//     Term 23 (AT2000-0250)/CC Outputs/Current setpoint value Ch.15 <-> Data Pointer/CurrentSetpointValues[14]
//     Term 23 (AT2000-0250)/CC Outputs/Current setpoint value Ch.2 <-> Data Pointer/CurrentSetpointValues[1]
//     Term 23 (AT2000-0250)/CC Outputs/Current setpoint value Ch.3 <-> Data Pointer/CurrentSetpointValues[2]
//     Term 23 (AT2000-0250)/CC Outputs/Current setpoint value Ch.4 <-> Data Pointer/CurrentSetpointValues[3]
//     Term 23 (AT2000-0250)/CC Outputs/Current setpoint value Ch.5 <-> Data Pointer/CurrentSetpointValues[4]
//     Term 23 (AT2000-0250)/CC Outputs/Current setpoint value Ch.6 <-> Data Pointer/CurrentSetpointValues[5]
//     Term 23 (AT2000-0250)/CC Outputs/Current setpoint value Ch.7 <-> Data Pointer/CurrentSetpointValues[6]
//     Term 23 (AT2000-0250)/CC Outputs/Current setpoint value Ch.8 <-> Data Pointer/CurrentSetpointValues[7]
//     Term 23 (AT2000-0250)/CC Outputs/Current setpoint value Ch.9 <-> Data Pointer/CurrentSetpointValues[8]
//     Term 23 (AT2000-0250)/Term 24 (AT2000-5250)/FB Inputs/Value Channel 01 <-> Data Pointer/RawPositionValues[0]
//     Term 23 (AT2000-0250)/Term 24 (AT2000-5250)/FB Inputs/Value Channel 02 <-> Data Pointer/RawPositionValues[1]
//     Term 23 (AT2000-0250)/Term 24 (AT2000-5250)/FB Inputs/Value Channel 03 <-> Data Pointer/RawPositionValues[2]
//     Term 23 (AT2000-0250)/Term 24 (AT2000-5250)/FB Inputs/Value Channel 04 <-> Data Pointer/RawPositionValues[3]
//     Term 23 (AT2000-0250)/Term 24 (AT2000-5250)/FB Inputs/Value Channel 05 <-> Data Pointer/RawPositionValues[4]
//     Term 23 (AT2000-0250)/Term 24 (AT2000-5250)/FB Inputs/Value Channel 06 <-> Data Pointer/RawPositionValues[5]
//     Term 23 (AT2000-0250)/Term 24 (AT2000-5250)/FB Inputs/Value Channel 07 <-> Data Pointer/RawPositionValues[6]
//     Term 23 (AT2000-0250)/Term 24 (AT2000-5250)/FB Inputs/Value Channel 08 <-> Data Pointer/RawPositionValues[7]
//     Term 23 (AT2000-0250)/Term 24 (AT2000-5250)/FB Inputs/Value Channel 09 <-> Data Pointer/RawPositionValues[8]
//     Term 23 (AT2000-0250)/Term 24 (AT2000-5250)/FB Inputs/Value Channel 10 <-> Data Pointer/RawPositionValues[9]
//     Term 23 (AT2000-0250)/Term 24 (AT2000-5250)/FB Inputs/Value Channel 11 <-> Data Pointer/RawPositionValues[10]
//     Term 23 (AT2000-0250)/Term 24 (AT2000-5250)/FB Inputs/Value Channel 12 <-> Data Pointer/RawPositionValues[11]
//     Term 23 (AT2000-0250)/Term 24 (AT2000-5250)/FB Inputs/Value Channel 13 <-> Data Pointer/RawPositionValues[12]
//     Term 23 (AT2000-0250)/Term 24 (AT2000-5250)/FB Inputs/Value Channel 14 <-> Data Pointer/RawPositionValues[13]
//     Term 23 (AT2000-0250)/Term 24 (AT2000-5250)/FB Inputs/Value Channel 15 <-> Data Pointer/RawPositionValues[14]
//     Term 23 (AT2000-0250)/Term 24 (AT2000-5250)/FB Inputs/Value Channel 16 <-> Data Pointer/RawPositionValues[15]
//     Term 23 (AT2000-0250)/Term 24 (AT2000-5250)/FB Inputs/Value Channel 17 <-> Data Pointer/RawPositionValues[16]
//     Term 23 (AT2000-0250)/Term 24 (AT2000-5250)/FB Inputs/Value Channel 18 <-> Data Pointer/RawPositionValues[17]
//     Term 23 (AT2000-0250)/Term 24 (AT2000-5250)/FB Inputs/Value Channel 19 <-> Data Pointer/RawPositionValues[18]
//     Term 23 (AT2000-0250)/Term 24 (AT2000-5250)/FB Inputs/Value Channel 20 <-> Data Pointer/RawPositionValues[19]
//     Term 23 (AT2000-0250)/Term 24 (AT2000-5250)/FB Inputs/Value Channel 21 <-> Data Pointer/RawPositionValues[20]
//     Term 23 (AT2000-0250)/Term 24 (AT2000-5250)/FB Inputs/Value Channel 22 <-> Data Pointer/RawPositionValues[21]
//     Term 23 (AT2000-0250)/Term 24 (AT2000-5250)/FB Inputs/Value Channel 23 <-> Data Pointer/RawPositionValues[22]
//     Term 23 (AT2000-0250)/Term 24 (AT2000-5250)/FB Inputs/Value Channel 24 <-> Data Pointer/RawPositionValues[23]
//     Term 23 (AT2000-0250)/Term 24 (AT2000-5250)/FB Inputs/Value Channel 25 <-> Data Pointer/RawPositionValues[24]
//     Term 23 (AT2000-0250)/Term 24 (AT2000-5250)/FB Inputs/Value Channel 26 <-> Data Pointer/RawPositionValues[25]
//     Term 23 (AT2000-0250)/Term 24 (AT2000-5250)/FB Inputs/Value Channel 27 <-> Data Pointer/RawPositionValues[26]
//     Term 23 (AT2000-0250)/Term 24 (AT2000-5250)/FB Inputs/Value Channel 28 <-> Data Pointer/RawPositionValues[27]
//     Term 23 (AT2000-0250)/Term 24 (AT2000-5250)/FB Inputs/Value Channel 29 <-> Data Pointer/RawPositionValues[28]
//     Term 23 (AT2000-0250)/Term 24 (AT2000-5250)/FB Inputs/Value Channel 30 <-> Data Pointer/RawPositionValues[29]
//     Term 23 (AT2000-0250)/Term 24 (AT2000-5250)/FB Inputs/Value Channel 31 <-> Data Pointer/RawPositionValues[30]
//     Term 23 (AT2000-0250)/Term 24 (AT2000-5250)/FB Inputs/Value Channel 32 <-> Data Pointer/RawPositionValues[31]
//   Device 16 <-> TcCOM Objects/XTS ProcessingUnit 1/Part 1/Module 7
//     Term 13 (AT2002-0250)/CC Inputs/Current actual value Ch.1 <-> Data Pointer/CurrentActualValues[0]
//     Term 13 (AT2002-0250)/CC Inputs/Current actual value Ch.10 <-> Data Pointer/CurrentActualValues[9]
//     Term 13 (AT2002-0250)/CC Inputs/Current actual value Ch.11 <-> Data Pointer/CurrentActualValues[10]
//     Term 13 (AT2002-0250)/CC Inputs/Current actual value Ch.12 <-> Data Pointer/CurrentActualValues[11]
//     Term 13 (AT2002-0250)/CC Inputs/Current actual value Ch.13 <-> Data Pointer/CurrentActualValues[12]
//     Term 13 (AT2002-0250)/CC Inputs/Current actual value Ch.14 <-> Data Pointer/CurrentActualValues[13]
//     Term 13 (AT2002-0250)/CC Inputs/Current actual value Ch.15 <-> Data Pointer/CurrentActualValues[14]
//     Term 13 (AT2002-0250)/CC Inputs/Current actual value Ch.2 <-> Data Pointer/CurrentActualValues[1]
//     Term 13 (AT2002-0250)/CC Inputs/Current actual value Ch.3 <-> Data Pointer/CurrentActualValues[2]
//     Term 13 (AT2002-0250)/CC Inputs/Current actual value Ch.4 <-> Data Pointer/CurrentActualValues[3]
//     Term 13 (AT2002-0250)/CC Inputs/Current actual value Ch.5 <-> Data Pointer/CurrentActualValues[4]
//     Term 13 (AT2002-0250)/CC Inputs/Current actual value Ch.6 <-> Data Pointer/CurrentActualValues[5]
//     Term 13 (AT2002-0250)/CC Inputs/Current actual value Ch.7 <-> Data Pointer/CurrentActualValues[6]
//     Term 13 (AT2002-0250)/CC Inputs/Current actual value Ch.8 <-> Data Pointer/CurrentActualValues[7]
//     Term 13 (AT2002-0250)/CC Inputs/Current actual value Ch.9 <-> Data Pointer/CurrentActualValues[8]
//     Term 13 (AT2002-0250)/CC Inputs/Status <-> Data Pointer/Status
//     Term 13 (AT2002-0250)/CC Outputs/Control <-> Data Pointer/Control
//     Term 13 (AT2002-0250)/CC Outputs/Current setpoint value Ch.1 <-> Data Pointer/CurrentSetpointValues[0]
//     Term 13 (AT2002-0250)/CC Outputs/Current setpoint value Ch.10 <-> Data Pointer/CurrentSetpointValues[9]
//     Term 13 (AT2002-0250)/CC Outputs/Current setpoint value Ch.11 <-> Data Pointer/CurrentSetpointValues[10]
//     Term 13 (AT2002-0250)/CC Outputs/Current setpoint value Ch.12 <-> Data Pointer/CurrentSetpointValues[11]
//     Term 13 (AT2002-0250)/CC Outputs/Current setpoint value Ch.13 <-> Data Pointer/CurrentSetpointValues[12]
//     Term 13 (AT2002-0250)/CC Outputs/Current setpoint value Ch.14 <-> Data Pointer/CurrentSetpointValues[13]
//     Term 13 (AT2002-0250)/CC Outputs/Current setpoint value Ch.15 <-> Data Pointer/CurrentSetpointValues[14]
//     Term 13 (AT2002-0250)/CC Outputs/Current setpoint value Ch.2 <-> Data Pointer/CurrentSetpointValues[1]
//     Term 13 (AT2002-0250)/CC Outputs/Current setpoint value Ch.3 <-> Data Pointer/CurrentSetpointValues[2]
//     Term 13 (AT2002-0250)/CC Outputs/Current setpoint value Ch.4 <-> Data Pointer/CurrentSetpointValues[3]
//     Term 13 (AT2002-0250)/CC Outputs/Current setpoint value Ch.5 <-> Data Pointer/CurrentSetpointValues[4]
//     Term 13 (AT2002-0250)/CC Outputs/Current setpoint value Ch.6 <-> Data Pointer/CurrentSetpointValues[5]
//     Term 13 (AT2002-0250)/CC Outputs/Current setpoint value Ch.7 <-> Data Pointer/CurrentSetpointValues[6]
//     Term 13 (AT2002-0250)/CC Outputs/Current setpoint value Ch.8 <-> Data Pointer/CurrentSetpointValues[7]
//     Term 13 (AT2002-0250)/CC Outputs/Current setpoint value Ch.9 <-> Data Pointer/CurrentSetpointValues[8]
//     Term 13 (AT2002-0250)/Term 14 (AT2002-5250)/FB Inputs/Value Channel 01 <-> Data Pointer/RawPositionValues[0]
//     Term 13 (AT2002-0250)/Term 14 (AT2002-5250)/FB Inputs/Value Channel 02 <-> Data Pointer/RawPositionValues[1]
//     Term 13 (AT2002-0250)/Term 14 (AT2002-5250)/FB Inputs/Value Channel 03 <-> Data Pointer/RawPositionValues[2]
//     Term 13 (AT2002-0250)/Term 14 (AT2002-5250)/FB Inputs/Value Channel 04 <-> Data Pointer/RawPositionValues[3]
//     Term 13 (AT2002-0250)/Term 14 (AT2002-5250)/FB Inputs/Value Channel 05 <-> Data Pointer/RawPositionValues[4]
//     Term 13 (AT2002-0250)/Term 14 (AT2002-5250)/FB Inputs/Value Channel 06 <-> Data Pointer/RawPositionValues[5]
//     Term 13 (AT2002-0250)/Term 14 (AT2002-5250)/FB Inputs/Value Channel 07 <-> Data Pointer/RawPositionValues[6]
//     Term 13 (AT2002-0250)/Term 14 (AT2002-5250)/FB Inputs/Value Channel 08 <-> Data Pointer/RawPositionValues[7]
//     Term 13 (AT2002-0250)/Term 14 (AT2002-5250)/FB Inputs/Value Channel 09 <-> Data Pointer/RawPositionValues[8]
//     Term 13 (AT2002-0250)/Term 14 (AT2002-5250)/FB Inputs/Value Channel 10 <-> Data Pointer/RawPositionValues[9]
//     Term 13 (AT2002-0250)/Term 14 (AT2002-5250)/FB Inputs/Value Channel 11 <-> Data Pointer/RawPositionValues[10]
//     Term 13 (AT2002-0250)/Term 14 (AT2002-5250)/FB Inputs/Value Channel 12 <-> Data Pointer/RawPositionValues[11]
//     Term 13 (AT2002-0250)/Term 14 (AT2002-5250)/FB Inputs/Value Channel 13 <-> Data Pointer/RawPositionValues[12]
//     Term 13 (AT2002-0250)/Term 14 (AT2002-5250)/FB Inputs/Value Channel 14 <-> Data Pointer/RawPositionValues[13]
//     Term 13 (AT2002-0250)/Term 14 (AT2002-5250)/FB Inputs/Value Channel 15 <-> Data Pointer/RawPositionValues[14]
//     Term 13 (AT2002-0250)/Term 14 (AT2002-5250)/FB Inputs/Value Channel 16 <-> Data Pointer/RawPositionValues[15]
//     Term 13 (AT2002-0250)/Term 14 (AT2002-5250)/FB Inputs/Value Channel 17 <-> Data Pointer/RawPositionValues[16]
//     Term 13 (AT2002-0250)/Term 14 (AT2002-5250)/FB Inputs/Value Channel 18 <-> Data Pointer/RawPositionValues[17]
//     Term 13 (AT2002-0250)/Term 14 (AT2002-5250)/FB Inputs/Value Channel 19 <-> Data Pointer/RawPositionValues[18]
//     Term 13 (AT2002-0250)/Term 14 (AT2002-5250)/FB Inputs/Value Channel 20 <-> Data Pointer/RawPositionValues[19]
//     Term 13 (AT2002-0250)/Term 14 (AT2002-5250)/FB Inputs/Value Channel 21 <-> Data Pointer/RawPositionValues[20]
//     Term 13 (AT2002-0250)/Term 14 (AT2002-5250)/FB Inputs/Value Channel 22 <-> Data Pointer/RawPositionValues[21]
//     Term 13 (AT2002-0250)/Term 14 (AT2002-5250)/FB Inputs/Value Channel 23 <-> Data Pointer/RawPositionValues[22]
//     Term 13 (AT2002-0250)/Term 14 (AT2002-5250)/FB Inputs/Value Channel 24 <-> Data Pointer/RawPositionValues[23]
//     Term 13 (AT2002-0250)/Term 14 (AT2002-5250)/FB Inputs/Value Channel 25 <-> Data Pointer/RawPositionValues[24]
//     Term 13 (AT2002-0250)/Term 14 (AT2002-5250)/FB Inputs/Value Channel 26 <-> Data Pointer/RawPositionValues[25]
//     Term 13 (AT2002-0250)/Term 14 (AT2002-5250)/FB Inputs/Value Channel 27 <-> Data Pointer/RawPositionValues[26]
//     Term 13 (AT2002-0250)/Term 14 (AT2002-5250)/FB Inputs/Value Channel 28 <-> Data Pointer/RawPositionValues[27]
//     Term 13 (AT2002-0250)/Term 14 (AT2002-5250)/FB Inputs/Value Channel 29 <-> Data Pointer/RawPositionValues[28]
//     Term 13 (AT2002-0250)/Term 14 (AT2002-5250)/FB Inputs/Value Channel 30 <-> Data Pointer/RawPositionValues[29]
//     Term 13 (AT2002-0250)/Term 14 (AT2002-5250)/FB Inputs/Value Channel 31 <-> Data Pointer/RawPositionValues[30]
//     Term 13 (AT2002-0250)/Term 14 (AT2002-5250)/FB Inputs/Value Channel 32 <-> Data Pointer/RawPositionValues[31]
//   Device 16 <-> TcCOM Objects/XTS ProcessingUnit 1/Part 1/Module 8
//     Term 15 (AT2000-0250)/CC Inputs/Current actual value Ch.1 <-> Data Pointer/CurrentActualValues[0]
//     Term 15 (AT2000-0250)/CC Inputs/Current actual value Ch.10 <-> Data Pointer/CurrentActualValues[9]
//     Term 15 (AT2000-0250)/CC Inputs/Current actual value Ch.11 <-> Data Pointer/CurrentActualValues[10]
//     Term 15 (AT2000-0250)/CC Inputs/Current actual value Ch.12 <-> Data Pointer/CurrentActualValues[11]
//     Term 15 (AT2000-0250)/CC Inputs/Current actual value Ch.13 <-> Data Pointer/CurrentActualValues[12]
//     Term 15 (AT2000-0250)/CC Inputs/Current actual value Ch.14 <-> Data Pointer/CurrentActualValues[13]
//     Term 15 (AT2000-0250)/CC Inputs/Current actual value Ch.15 <-> Data Pointer/CurrentActualValues[14]
//     Term 15 (AT2000-0250)/CC Inputs/Current actual value Ch.2 <-> Data Pointer/CurrentActualValues[1]
//     Term 15 (AT2000-0250)/CC Inputs/Current actual value Ch.3 <-> Data Pointer/CurrentActualValues[2]
//     Term 15 (AT2000-0250)/CC Inputs/Current actual value Ch.4 <-> Data Pointer/CurrentActualValues[3]
//     Term 15 (AT2000-0250)/CC Inputs/Current actual value Ch.5 <-> Data Pointer/CurrentActualValues[4]
//     Term 15 (AT2000-0250)/CC Inputs/Current actual value Ch.6 <-> Data Pointer/CurrentActualValues[5]
//     Term 15 (AT2000-0250)/CC Inputs/Current actual value Ch.7 <-> Data Pointer/CurrentActualValues[6]
//     Term 15 (AT2000-0250)/CC Inputs/Current actual value Ch.8 <-> Data Pointer/CurrentActualValues[7]
//     Term 15 (AT2000-0250)/CC Inputs/Current actual value Ch.9 <-> Data Pointer/CurrentActualValues[8]
//     Term 15 (AT2000-0250)/CC Inputs/Status <-> Data Pointer/Status
//     Term 15 (AT2000-0250)/CC Outputs/Control <-> Data Pointer/Control
//     Term 15 (AT2000-0250)/CC Outputs/Current setpoint value Ch.1 <-> Data Pointer/CurrentSetpointValues[0]
//     Term 15 (AT2000-0250)/CC Outputs/Current setpoint value Ch.10 <-> Data Pointer/CurrentSetpointValues[9]
//     Term 15 (AT2000-0250)/CC Outputs/Current setpoint value Ch.11 <-> Data Pointer/CurrentSetpointValues[10]
//     Term 15 (AT2000-0250)/CC Outputs/Current setpoint value Ch.12 <-> Data Pointer/CurrentSetpointValues[11]
//     Term 15 (AT2000-0250)/CC Outputs/Current setpoint value Ch.13 <-> Data Pointer/CurrentSetpointValues[12]
//     Term 15 (AT2000-0250)/CC Outputs/Current setpoint value Ch.14 <-> Data Pointer/CurrentSetpointValues[13]
//     Term 15 (AT2000-0250)/CC Outputs/Current setpoint value Ch.15 <-> Data Pointer/CurrentSetpointValues[14]
//     Term 15 (AT2000-0250)/CC Outputs/Current setpoint value Ch.2 <-> Data Pointer/CurrentSetpointValues[1]
//     Term 15 (AT2000-0250)/CC Outputs/Current setpoint value Ch.3 <-> Data Pointer/CurrentSetpointValues[2]
//     Term 15 (AT2000-0250)/CC Outputs/Current setpoint value Ch.4 <-> Data Pointer/CurrentSetpointValues[3]
//     Term 15 (AT2000-0250)/CC Outputs/Current setpoint value Ch.5 <-> Data Pointer/CurrentSetpointValues[4]
//     Term 15 (AT2000-0250)/CC Outputs/Current setpoint value Ch.6 <-> Data Pointer/CurrentSetpointValues[5]
//     Term 15 (AT2000-0250)/CC Outputs/Current setpoint value Ch.7 <-> Data Pointer/CurrentSetpointValues[6]
//     Term 15 (AT2000-0250)/CC Outputs/Current setpoint value Ch.8 <-> Data Pointer/CurrentSetpointValues[7]
//     Term 15 (AT2000-0250)/CC Outputs/Current setpoint value Ch.9 <-> Data Pointer/CurrentSetpointValues[8]
//     Term 15 (AT2000-0250)/Term 16 (AT2000-5250)/FB Inputs/Value Channel 01 <-> Data Pointer/RawPositionValues[0]
//     Term 15 (AT2000-0250)/Term 16 (AT2000-5250)/FB Inputs/Value Channel 02 <-> Data Pointer/RawPositionValues[1]
//     Term 15 (AT2000-0250)/Term 16 (AT2000-5250)/FB Inputs/Value Channel 03 <-> Data Pointer/RawPositionValues[2]
//     Term 15 (AT2000-0250)/Term 16 (AT2000-5250)/FB Inputs/Value Channel 04 <-> Data Pointer/RawPositionValues[3]
//     Term 15 (AT2000-0250)/Term 16 (AT2000-5250)/FB Inputs/Value Channel 05 <-> Data Pointer/RawPositionValues[4]
//     Term 15 (AT2000-0250)/Term 16 (AT2000-5250)/FB Inputs/Value Channel 06 <-> Data Pointer/RawPositionValues[5]
//     Term 15 (AT2000-0250)/Term 16 (AT2000-5250)/FB Inputs/Value Channel 07 <-> Data Pointer/RawPositionValues[6]
//     Term 15 (AT2000-0250)/Term 16 (AT2000-5250)/FB Inputs/Value Channel 08 <-> Data Pointer/RawPositionValues[7]
//     Term 15 (AT2000-0250)/Term 16 (AT2000-5250)/FB Inputs/Value Channel 09 <-> Data Pointer/RawPositionValues[8]
//     Term 15 (AT2000-0250)/Term 16 (AT2000-5250)/FB Inputs/Value Channel 10 <-> Data Pointer/RawPositionValues[9]
//     Term 15 (AT2000-0250)/Term 16 (AT2000-5250)/FB Inputs/Value Channel 11 <-> Data Pointer/RawPositionValues[10]
//     Term 15 (AT2000-0250)/Term 16 (AT2000-5250)/FB Inputs/Value Channel 12 <-> Data Pointer/RawPositionValues[11]
//     Term 15 (AT2000-0250)/Term 16 (AT2000-5250)/FB Inputs/Value Channel 13 <-> Data Pointer/RawPositionValues[12]
//     Term 15 (AT2000-0250)/Term 16 (AT2000-5250)/FB Inputs/Value Channel 14 <-> Data Pointer/RawPositionValues[13]
//     Term 15 (AT2000-0250)/Term 16 (AT2000-5250)/FB Inputs/Value Channel 15 <-> Data Pointer/RawPositionValues[14]
//     Term 15 (AT2000-0250)/Term 16 (AT2000-5250)/FB Inputs/Value Channel 16 <-> Data Pointer/RawPositionValues[15]
//     Term 15 (AT2000-0250)/Term 16 (AT2000-5250)/FB Inputs/Value Channel 17 <-> Data Pointer/RawPositionValues[16]
//     Term 15 (AT2000-0250)/Term 16 (AT2000-5250)/FB Inputs/Value Channel 18 <-> Data Pointer/RawPositionValues[17]
//     Term 15 (AT2000-0250)/Term 16 (AT2000-5250)/FB Inputs/Value Channel 19 <-> Data Pointer/RawPositionValues[18]
//     Term 15 (AT2000-0250)/Term 16 (AT2000-5250)/FB Inputs/Value Channel 20 <-> Data Pointer/RawPositionValues[19]
//     Term 15 (AT2000-0250)/Term 16 (AT2000-5250)/FB Inputs/Value Channel 21 <-> Data Pointer/RawPositionValues[20]
//     Term 15 (AT2000-0250)/Term 16 (AT2000-5250)/FB Inputs/Value Channel 22 <-> Data Pointer/RawPositionValues[21]
//     Term 15 (AT2000-0250)/Term 16 (AT2000-5250)/FB Inputs/Value Channel 23 <-> Data Pointer/RawPositionValues[22]
//     Term 15 (AT2000-0250)/Term 16 (AT2000-5250)/FB Inputs/Value Channel 24 <-> Data Pointer/RawPositionValues[23]
//     Term 15 (AT2000-0250)/Term 16 (AT2000-5250)/FB Inputs/Value Channel 25 <-> Data Pointer/RawPositionValues[24]
//     Term 15 (AT2000-0250)/Term 16 (AT2000-5250)/FB Inputs/Value Channel 26 <-> Data Pointer/RawPositionValues[25]
//     Term 15 (AT2000-0250)/Term 16 (AT2000-5250)/FB Inputs/Value Channel 27 <-> Data Pointer/RawPositionValues[26]
//     Term 15 (AT2000-0250)/Term 16 (AT2000-5250)/FB Inputs/Value Channel 28 <-> Data Pointer/RawPositionValues[27]
//     Term 15 (AT2000-0250)/Term 16 (AT2000-5250)/FB Inputs/Value Channel 29 <-> Data Pointer/RawPositionValues[28]
//     Term 15 (AT2000-0250)/Term 16 (AT2000-5250)/FB Inputs/Value Channel 30 <-> Data Pointer/RawPositionValues[29]
//     Term 15 (AT2000-0250)/Term 16 (AT2000-5250)/FB Inputs/Value Channel 31 <-> Data Pointer/RawPositionValues[30]
//     Term 15 (AT2000-0250)/Term 16 (AT2000-5250)/FB Inputs/Value Channel 32 <-> Data Pointer/RawPositionValues[31]
//   Device 16 <-> TcCOM Objects/XTS ProcessingUnit 1/Part 1/Module 9
//     Term 17 (AT2000-0250)/CC Inputs/Current actual value Ch.1 <-> Data Pointer/CurrentActualValues[0]
//     Term 17 (AT2000-0250)/CC Inputs/Current actual value Ch.10 <-> Data Pointer/CurrentActualValues[9]
//     Term 17 (AT2000-0250)/CC Inputs/Current actual value Ch.11 <-> Data Pointer/CurrentActualValues[10]
//     Term 17 (AT2000-0250)/CC Inputs/Current actual value Ch.12 <-> Data Pointer/CurrentActualValues[11]
//     Term 17 (AT2000-0250)/CC Inputs/Current actual value Ch.13 <-> Data Pointer/CurrentActualValues[12]
//     Term 17 (AT2000-0250)/CC Inputs/Current actual value Ch.14 <-> Data Pointer/CurrentActualValues[13]
//     Term 17 (AT2000-0250)/CC Inputs/Current actual value Ch.15 <-> Data Pointer/CurrentActualValues[14]
//     Term 17 (AT2000-0250)/CC Inputs/Current actual value Ch.2 <-> Data Pointer/CurrentActualValues[1]
//     Term 17 (AT2000-0250)/CC Inputs/Current actual value Ch.3 <-> Data Pointer/CurrentActualValues[2]
//     Term 17 (AT2000-0250)/CC Inputs/Current actual value Ch.4 <-> Data Pointer/CurrentActualValues[3]
//     Term 17 (AT2000-0250)/CC Inputs/Current actual value Ch.5 <-> Data Pointer/CurrentActualValues[4]
//     Term 17 (AT2000-0250)/CC Inputs/Current actual value Ch.6 <-> Data Pointer/CurrentActualValues[5]
//     Term 17 (AT2000-0250)/CC Inputs/Current actual value Ch.7 <-> Data Pointer/CurrentActualValues[6]
//     Term 17 (AT2000-0250)/CC Inputs/Current actual value Ch.8 <-> Data Pointer/CurrentActualValues[7]
//     Term 17 (AT2000-0250)/CC Inputs/Current actual value Ch.9 <-> Data Pointer/CurrentActualValues[8]
//     Term 17 (AT2000-0250)/CC Inputs/Status <-> Data Pointer/Status
//     Term 17 (AT2000-0250)/CC Outputs/Control <-> Data Pointer/Control
//     Term 17 (AT2000-0250)/CC Outputs/Current setpoint value Ch.1 <-> Data Pointer/CurrentSetpointValues[0]
//     Term 17 (AT2000-0250)/CC Outputs/Current setpoint value Ch.10 <-> Data Pointer/CurrentSetpointValues[9]
//     Term 17 (AT2000-0250)/CC Outputs/Current setpoint value Ch.11 <-> Data Pointer/CurrentSetpointValues[10]
//     Term 17 (AT2000-0250)/CC Outputs/Current setpoint value Ch.12 <-> Data Pointer/CurrentSetpointValues[11]
//     Term 17 (AT2000-0250)/CC Outputs/Current setpoint value Ch.13 <-> Data Pointer/CurrentSetpointValues[12]
//     Term 17 (AT2000-0250)/CC Outputs/Current setpoint value Ch.14 <-> Data Pointer/CurrentSetpointValues[13]
//     Term 17 (AT2000-0250)/CC Outputs/Current setpoint value Ch.15 <-> Data Pointer/CurrentSetpointValues[14]
//     Term 17 (AT2000-0250)/CC Outputs/Current setpoint value Ch.2 <-> Data Pointer/CurrentSetpointValues[1]
//     Term 17 (AT2000-0250)/CC Outputs/Current setpoint value Ch.3 <-> Data Pointer/CurrentSetpointValues[2]
//     Term 17 (AT2000-0250)/CC Outputs/Current setpoint value Ch.4 <-> Data Pointer/CurrentSetpointValues[3]
//     Term 17 (AT2000-0250)/CC Outputs/Current setpoint value Ch.5 <-> Data Pointer/CurrentSetpointValues[4]
//     Term 17 (AT2000-0250)/CC Outputs/Current setpoint value Ch.6 <-> Data Pointer/CurrentSetpointValues[5]
//     Term 17 (AT2000-0250)/CC Outputs/Current setpoint value Ch.7 <-> Data Pointer/CurrentSetpointValues[6]
//     Term 17 (AT2000-0250)/CC Outputs/Current setpoint value Ch.8 <-> Data Pointer/CurrentSetpointValues[7]
//     Term 17 (AT2000-0250)/CC Outputs/Current setpoint value Ch.9 <-> Data Pointer/CurrentSetpointValues[8]
//     Term 17 (AT2000-0250)/Term 18 (AT2000-5250)/FB Inputs/Value Channel 01 <-> Data Pointer/RawPositionValues[0]
//     Term 17 (AT2000-0250)/Term 18 (AT2000-5250)/FB Inputs/Value Channel 02 <-> Data Pointer/RawPositionValues[1]
//     Term 17 (AT2000-0250)/Term 18 (AT2000-5250)/FB Inputs/Value Channel 03 <-> Data Pointer/RawPositionValues[2]
//     Term 17 (AT2000-0250)/Term 18 (AT2000-5250)/FB Inputs/Value Channel 04 <-> Data Pointer/RawPositionValues[3]
//     Term 17 (AT2000-0250)/Term 18 (AT2000-5250)/FB Inputs/Value Channel 05 <-> Data Pointer/RawPositionValues[4]
//     Term 17 (AT2000-0250)/Term 18 (AT2000-5250)/FB Inputs/Value Channel 06 <-> Data Pointer/RawPositionValues[5]
//     Term 17 (AT2000-0250)/Term 18 (AT2000-5250)/FB Inputs/Value Channel 07 <-> Data Pointer/RawPositionValues[6]
//     Term 17 (AT2000-0250)/Term 18 (AT2000-5250)/FB Inputs/Value Channel 08 <-> Data Pointer/RawPositionValues[7]
//     Term 17 (AT2000-0250)/Term 18 (AT2000-5250)/FB Inputs/Value Channel 09 <-> Data Pointer/RawPositionValues[8]
//     Term 17 (AT2000-0250)/Term 18 (AT2000-5250)/FB Inputs/Value Channel 10 <-> Data Pointer/RawPositionValues[9]
//     Term 17 (AT2000-0250)/Term 18 (AT2000-5250)/FB Inputs/Value Channel 11 <-> Data Pointer/RawPositionValues[10]
//     Term 17 (AT2000-0250)/Term 18 (AT2000-5250)/FB Inputs/Value Channel 12 <-> Data Pointer/RawPositionValues[11]
//     Term 17 (AT2000-0250)/Term 18 (AT2000-5250)/FB Inputs/Value Channel 13 <-> Data Pointer/RawPositionValues[12]
//     Term 17 (AT2000-0250)/Term 18 (AT2000-5250)/FB Inputs/Value Channel 14 <-> Data Pointer/RawPositionValues[13]
//     Term 17 (AT2000-0250)/Term 18 (AT2000-5250)/FB Inputs/Value Channel 15 <-> Data Pointer/RawPositionValues[14]
//     Term 17 (AT2000-0250)/Term 18 (AT2000-5250)/FB Inputs/Value Channel 16 <-> Data Pointer/RawPositionValues[15]
//     Term 17 (AT2000-0250)/Term 18 (AT2000-5250)/FB Inputs/Value Channel 17 <-> Data Pointer/RawPositionValues[16]
//     Term 17 (AT2000-0250)/Term 18 (AT2000-5250)/FB Inputs/Value Channel 18 <-> Data Pointer/RawPositionValues[17]
//     Term 17 (AT2000-0250)/Term 18 (AT2000-5250)/FB Inputs/Value Channel 19 <-> Data Pointer/RawPositionValues[18]
//     Term 17 (AT2000-0250)/Term 18 (AT2000-5250)/FB Inputs/Value Channel 20 <-> Data Pointer/RawPositionValues[19]
//     Term 17 (AT2000-0250)/Term 18 (AT2000-5250)/FB Inputs/Value Channel 21 <-> Data Pointer/RawPositionValues[20]
//     Term 17 (AT2000-0250)/Term 18 (AT2000-5250)/FB Inputs/Value Channel 22 <-> Data Pointer/RawPositionValues[21]
//     Term 17 (AT2000-0250)/Term 18 (AT2000-5250)/FB Inputs/Value Channel 23 <-> Data Pointer/RawPositionValues[22]
//     Term 17 (AT2000-0250)/Term 18 (AT2000-5250)/FB Inputs/Value Channel 24 <-> Data Pointer/RawPositionValues[23]
//     Term 17 (AT2000-0250)/Term 18 (AT2000-5250)/FB Inputs/Value Channel 25 <-> Data Pointer/RawPositionValues[24]
//     Term 17 (AT2000-0250)/Term 18 (AT2000-5250)/FB Inputs/Value Channel 26 <-> Data Pointer/RawPositionValues[25]
//     Term 17 (AT2000-0250)/Term 18 (AT2000-5250)/FB Inputs/Value Channel 27 <-> Data Pointer/RawPositionValues[26]
//     Term 17 (AT2000-0250)/Term 18 (AT2000-5250)/FB Inputs/Value Channel 28 <-> Data Pointer/RawPositionValues[27]
//     Term 17 (AT2000-0250)/Term 18 (AT2000-5250)/FB Inputs/Value Channel 29 <-> Data Pointer/RawPositionValues[28]
//     Term 17 (AT2000-0250)/Term 18 (AT2000-5250)/FB Inputs/Value Channel 30 <-> Data Pointer/RawPositionValues[29]
//     Term 17 (AT2000-0250)/Term 18 (AT2000-5250)/FB Inputs/Value Channel 31 <-> Data Pointer/RawPositionValues[30]
//     Term 17 (AT2000-0250)/Term 18 (AT2000-5250)/FB Inputs/Value Channel 32 <-> Data Pointer/RawPositionValues[31]
//   Device 17 <-> TcCOM Objects/XTS ProcessingUnit 1/Part 1/Module 13
//     Term 25 (AT2002-0250)/CC Inputs/Current actual value Ch.1 <-> Data Pointer/CurrentActualValues[0]
//     Term 25 (AT2002-0250)/CC Inputs/Current actual value Ch.10 <-> Data Pointer/CurrentActualValues[9]
//     Term 25 (AT2002-0250)/CC Inputs/Current actual value Ch.11 <-> Data Pointer/CurrentActualValues[10]
//     Term 25 (AT2002-0250)/CC Inputs/Current actual value Ch.12 <-> Data Pointer/CurrentActualValues[11]
//     Term 25 (AT2002-0250)/CC Inputs/Current actual value Ch.13 <-> Data Pointer/CurrentActualValues[12]
//     Term 25 (AT2002-0250)/CC Inputs/Current actual value Ch.14 <-> Data Pointer/CurrentActualValues[13]
//     Term 25 (AT2002-0250)/CC Inputs/Current actual value Ch.15 <-> Data Pointer/CurrentActualValues[14]
//     Term 25 (AT2002-0250)/CC Inputs/Current actual value Ch.2 <-> Data Pointer/CurrentActualValues[1]
//     Term 25 (AT2002-0250)/CC Inputs/Current actual value Ch.3 <-> Data Pointer/CurrentActualValues[2]
//     Term 25 (AT2002-0250)/CC Inputs/Current actual value Ch.4 <-> Data Pointer/CurrentActualValues[3]
//     Term 25 (AT2002-0250)/CC Inputs/Current actual value Ch.5 <-> Data Pointer/CurrentActualValues[4]
//     Term 25 (AT2002-0250)/CC Inputs/Current actual value Ch.6 <-> Data Pointer/CurrentActualValues[5]
//     Term 25 (AT2002-0250)/CC Inputs/Current actual value Ch.7 <-> Data Pointer/CurrentActualValues[6]
//     Term 25 (AT2002-0250)/CC Inputs/Current actual value Ch.8 <-> Data Pointer/CurrentActualValues[7]
//     Term 25 (AT2002-0250)/CC Inputs/Current actual value Ch.9 <-> Data Pointer/CurrentActualValues[8]
//     Term 25 (AT2002-0250)/CC Inputs/Status <-> Data Pointer/Status
//     Term 25 (AT2002-0250)/CC Outputs/Control <-> Data Pointer/Control
//     Term 25 (AT2002-0250)/CC Outputs/Current setpoint value Ch.1 <-> Data Pointer/CurrentSetpointValues[0]
//     Term 25 (AT2002-0250)/CC Outputs/Current setpoint value Ch.10 <-> Data Pointer/CurrentSetpointValues[9]
//     Term 25 (AT2002-0250)/CC Outputs/Current setpoint value Ch.11 <-> Data Pointer/CurrentSetpointValues[10]
//     Term 25 (AT2002-0250)/CC Outputs/Current setpoint value Ch.12 <-> Data Pointer/CurrentSetpointValues[11]
//     Term 25 (AT2002-0250)/CC Outputs/Current setpoint value Ch.13 <-> Data Pointer/CurrentSetpointValues[12]
//     Term 25 (AT2002-0250)/CC Outputs/Current setpoint value Ch.14 <-> Data Pointer/CurrentSetpointValues[13]
//     Term 25 (AT2002-0250)/CC Outputs/Current setpoint value Ch.15 <-> Data Pointer/CurrentSetpointValues[14]
//     Term 25 (AT2002-0250)/CC Outputs/Current setpoint value Ch.2 <-> Data Pointer/CurrentSetpointValues[1]
//     Term 25 (AT2002-0250)/CC Outputs/Current setpoint value Ch.3 <-> Data Pointer/CurrentSetpointValues[2]
//     Term 25 (AT2002-0250)/CC Outputs/Current setpoint value Ch.4 <-> Data Pointer/CurrentSetpointValues[3]
//     Term 25 (AT2002-0250)/CC Outputs/Current setpoint value Ch.5 <-> Data Pointer/CurrentSetpointValues[4]
//     Term 25 (AT2002-0250)/CC Outputs/Current setpoint value Ch.6 <-> Data Pointer/CurrentSetpointValues[5]
//     Term 25 (AT2002-0250)/CC Outputs/Current setpoint value Ch.7 <-> Data Pointer/CurrentSetpointValues[6]
//     Term 25 (AT2002-0250)/CC Outputs/Current setpoint value Ch.8 <-> Data Pointer/CurrentSetpointValues[7]
//     Term 25 (AT2002-0250)/CC Outputs/Current setpoint value Ch.9 <-> Data Pointer/CurrentSetpointValues[8]
//     Term 25 (AT2002-0250)/Term 26 (AT2002-5250)/FB Inputs/Value Channel 01 <-> Data Pointer/RawPositionValues[0]
//     Term 25 (AT2002-0250)/Term 26 (AT2002-5250)/FB Inputs/Value Channel 02 <-> Data Pointer/RawPositionValues[1]
//     Term 25 (AT2002-0250)/Term 26 (AT2002-5250)/FB Inputs/Value Channel 03 <-> Data Pointer/RawPositionValues[2]
//     Term 25 (AT2002-0250)/Term 26 (AT2002-5250)/FB Inputs/Value Channel 04 <-> Data Pointer/RawPositionValues[3]
//     Term 25 (AT2002-0250)/Term 26 (AT2002-5250)/FB Inputs/Value Channel 05 <-> Data Pointer/RawPositionValues[4]
//     Term 25 (AT2002-0250)/Term 26 (AT2002-5250)/FB Inputs/Value Channel 06 <-> Data Pointer/RawPositionValues[5]
//     Term 25 (AT2002-0250)/Term 26 (AT2002-5250)/FB Inputs/Value Channel 07 <-> Data Pointer/RawPositionValues[6]
//     Term 25 (AT2002-0250)/Term 26 (AT2002-5250)/FB Inputs/Value Channel 08 <-> Data Pointer/RawPositionValues[7]
//     Term 25 (AT2002-0250)/Term 26 (AT2002-5250)/FB Inputs/Value Channel 09 <-> Data Pointer/RawPositionValues[8]
//     Term 25 (AT2002-0250)/Term 26 (AT2002-5250)/FB Inputs/Value Channel 10 <-> Data Pointer/RawPositionValues[9]
//     Term 25 (AT2002-0250)/Term 26 (AT2002-5250)/FB Inputs/Value Channel 11 <-> Data Pointer/RawPositionValues[10]
//     Term 25 (AT2002-0250)/Term 26 (AT2002-5250)/FB Inputs/Value Channel 12 <-> Data Pointer/RawPositionValues[11]
//     Term 25 (AT2002-0250)/Term 26 (AT2002-5250)/FB Inputs/Value Channel 13 <-> Data Pointer/RawPositionValues[12]
//     Term 25 (AT2002-0250)/Term 26 (AT2002-5250)/FB Inputs/Value Channel 14 <-> Data Pointer/RawPositionValues[13]
//     Term 25 (AT2002-0250)/Term 26 (AT2002-5250)/FB Inputs/Value Channel 15 <-> Data Pointer/RawPositionValues[14]
//     Term 25 (AT2002-0250)/Term 26 (AT2002-5250)/FB Inputs/Value Channel 16 <-> Data Pointer/RawPositionValues[15]
//     Term 25 (AT2002-0250)/Term 26 (AT2002-5250)/FB Inputs/Value Channel 17 <-> Data Pointer/RawPositionValues[16]
//     Term 25 (AT2002-0250)/Term 26 (AT2002-5250)/FB Inputs/Value Channel 18 <-> Data Pointer/RawPositionValues[17]
//     Term 25 (AT2002-0250)/Term 26 (AT2002-5250)/FB Inputs/Value Channel 19 <-> Data Pointer/RawPositionValues[18]
//     Term 25 (AT2002-0250)/Term 26 (AT2002-5250)/FB Inputs/Value Channel 20 <-> Data Pointer/RawPositionValues[19]
//     Term 25 (AT2002-0250)/Term 26 (AT2002-5250)/FB Inputs/Value Channel 21 <-> Data Pointer/RawPositionValues[20]
//     Term 25 (AT2002-0250)/Term 26 (AT2002-5250)/FB Inputs/Value Channel 22 <-> Data Pointer/RawPositionValues[21]
//     Term 25 (AT2002-0250)/Term 26 (AT2002-5250)/FB Inputs/Value Channel 23 <-> Data Pointer/RawPositionValues[22]
//     Term 25 (AT2002-0250)/Term 26 (AT2002-5250)/FB Inputs/Value Channel 24 <-> Data Pointer/RawPositionValues[23]
//     Term 25 (AT2002-0250)/Term 26 (AT2002-5250)/FB Inputs/Value Channel 25 <-> Data Pointer/RawPositionValues[24]
//     Term 25 (AT2002-0250)/Term 26 (AT2002-5250)/FB Inputs/Value Channel 26 <-> Data Pointer/RawPositionValues[25]
//     Term 25 (AT2002-0250)/Term 26 (AT2002-5250)/FB Inputs/Value Channel 27 <-> Data Pointer/RawPositionValues[26]
//     Term 25 (AT2002-0250)/Term 26 (AT2002-5250)/FB Inputs/Value Channel 28 <-> Data Pointer/RawPositionValues[27]
//     Term 25 (AT2002-0250)/Term 26 (AT2002-5250)/FB Inputs/Value Channel 29 <-> Data Pointer/RawPositionValues[28]
//     Term 25 (AT2002-0250)/Term 26 (AT2002-5250)/FB Inputs/Value Channel 30 <-> Data Pointer/RawPositionValues[29]
//     Term 25 (AT2002-0250)/Term 26 (AT2002-5250)/FB Inputs/Value Channel 31 <-> Data Pointer/RawPositionValues[30]
//     Term 25 (AT2002-0250)/Term 26 (AT2002-5250)/FB Inputs/Value Channel 32 <-> Data Pointer/RawPositionValues[31]
//   Device 17 <-> TcCOM Objects/XTS ProcessingUnit 1/Part 1/Module 14
//     Term 27 (AT2000-0250)/CC Inputs/Current actual value Ch.1 <-> Data Pointer/CurrentActualValues[0]
//     Term 27 (AT2000-0250)/CC Inputs/Current actual value Ch.10 <-> Data Pointer/CurrentActualValues[9]
//     Term 27 (AT2000-0250)/CC Inputs/Current actual value Ch.11 <-> Data Pointer/CurrentActualValues[10]
//     Term 27 (AT2000-0250)/CC Inputs/Current actual value Ch.12 <-> Data Pointer/CurrentActualValues[11]
//     Term 27 (AT2000-0250)/CC Inputs/Current actual value Ch.13 <-> Data Pointer/CurrentActualValues[12]
//     Term 27 (AT2000-0250)/CC Inputs/Current actual value Ch.14 <-> Data Pointer/CurrentActualValues[13]
//     Term 27 (AT2000-0250)/CC Inputs/Current actual value Ch.15 <-> Data Pointer/CurrentActualValues[14]
//     Term 27 (AT2000-0250)/CC Inputs/Current actual value Ch.2 <-> Data Pointer/CurrentActualValues[1]
//     Term 27 (AT2000-0250)/CC Inputs/Current actual value Ch.3 <-> Data Pointer/CurrentActualValues[2]
//     Term 27 (AT2000-0250)/CC Inputs/Current actual value Ch.4 <-> Data Pointer/CurrentActualValues[3]
//     Term 27 (AT2000-0250)/CC Inputs/Current actual value Ch.5 <-> Data Pointer/CurrentActualValues[4]
//     Term 27 (AT2000-0250)/CC Inputs/Current actual value Ch.6 <-> Data Pointer/CurrentActualValues[5]
//     Term 27 (AT2000-0250)/CC Inputs/Current actual value Ch.7 <-> Data Pointer/CurrentActualValues[6]
//     Term 27 (AT2000-0250)/CC Inputs/Current actual value Ch.8 <-> Data Pointer/CurrentActualValues[7]
//     Term 27 (AT2000-0250)/CC Inputs/Current actual value Ch.9 <-> Data Pointer/CurrentActualValues[8]
//     Term 27 (AT2000-0250)/CC Inputs/Status <-> Data Pointer/Status
//     Term 27 (AT2000-0250)/CC Outputs/Control <-> Data Pointer/Control
//     Term 27 (AT2000-0250)/CC Outputs/Current setpoint value Ch.1 <-> Data Pointer/CurrentSetpointValues[0]
//     Term 27 (AT2000-0250)/CC Outputs/Current setpoint value Ch.10 <-> Data Pointer/CurrentSetpointValues[9]
//     Term 27 (AT2000-0250)/CC Outputs/Current setpoint value Ch.11 <-> Data Pointer/CurrentSetpointValues[10]
//     Term 27 (AT2000-0250)/CC Outputs/Current setpoint value Ch.12 <-> Data Pointer/CurrentSetpointValues[11]
//     Term 27 (AT2000-0250)/CC Outputs/Current setpoint value Ch.13 <-> Data Pointer/CurrentSetpointValues[12]
//     Term 27 (AT2000-0250)/CC Outputs/Current setpoint value Ch.14 <-> Data Pointer/CurrentSetpointValues[13]
//     Term 27 (AT2000-0250)/CC Outputs/Current setpoint value Ch.15 <-> Data Pointer/CurrentSetpointValues[14]
//     Term 27 (AT2000-0250)/CC Outputs/Current setpoint value Ch.2 <-> Data Pointer/CurrentSetpointValues[1]
//     Term 27 (AT2000-0250)/CC Outputs/Current setpoint value Ch.3 <-> Data Pointer/CurrentSetpointValues[2]
//     Term 27 (AT2000-0250)/CC Outputs/Current setpoint value Ch.4 <-> Data Pointer/CurrentSetpointValues[3]
//     Term 27 (AT2000-0250)/CC Outputs/Current setpoint value Ch.5 <-> Data Pointer/CurrentSetpointValues[4]
//     Term 27 (AT2000-0250)/CC Outputs/Current setpoint value Ch.6 <-> Data Pointer/CurrentSetpointValues[5]
//     Term 27 (AT2000-0250)/CC Outputs/Current setpoint value Ch.7 <-> Data Pointer/CurrentSetpointValues[6]
//     Term 27 (AT2000-0250)/CC Outputs/Current setpoint value Ch.8 <-> Data Pointer/CurrentSetpointValues[7]
//     Term 27 (AT2000-0250)/CC Outputs/Current setpoint value Ch.9 <-> Data Pointer/CurrentSetpointValues[8]
//     Term 27 (AT2000-0250)/Term 28 (AT2000-5250)/FB Inputs/Value Channel 01 <-> Data Pointer/RawPositionValues[0]
//     Term 27 (AT2000-0250)/Term 28 (AT2000-5250)/FB Inputs/Value Channel 02 <-> Data Pointer/RawPositionValues[1]
//     Term 27 (AT2000-0250)/Term 28 (AT2000-5250)/FB Inputs/Value Channel 03 <-> Data Pointer/RawPositionValues[2]
//     Term 27 (AT2000-0250)/Term 28 (AT2000-5250)/FB Inputs/Value Channel 04 <-> Data Pointer/RawPositionValues[3]
//     Term 27 (AT2000-0250)/Term 28 (AT2000-5250)/FB Inputs/Value Channel 05 <-> Data Pointer/RawPositionValues[4]
//     Term 27 (AT2000-0250)/Term 28 (AT2000-5250)/FB Inputs/Value Channel 06 <-> Data Pointer/RawPositionValues[5]
//     Term 27 (AT2000-0250)/Term 28 (AT2000-5250)/FB Inputs/Value Channel 07 <-> Data Pointer/RawPositionValues[6]
//     Term 27 (AT2000-0250)/Term 28 (AT2000-5250)/FB Inputs/Value Channel 08 <-> Data Pointer/RawPositionValues[7]
//     Term 27 (AT2000-0250)/Term 28 (AT2000-5250)/FB Inputs/Value Channel 09 <-> Data Pointer/RawPositionValues[8]
//     Term 27 (AT2000-0250)/Term 28 (AT2000-5250)/FB Inputs/Value Channel 10 <-> Data Pointer/RawPositionValues[9]
//     Term 27 (AT2000-0250)/Term 28 (AT2000-5250)/FB Inputs/Value Channel 11 <-> Data Pointer/RawPositionValues[10]
//     Term 27 (AT2000-0250)/Term 28 (AT2000-5250)/FB Inputs/Value Channel 12 <-> Data Pointer/RawPositionValues[11]
//     Term 27 (AT2000-0250)/Term 28 (AT2000-5250)/FB Inputs/Value Channel 13 <-> Data Pointer/RawPositionValues[12]
//     Term 27 (AT2000-0250)/Term 28 (AT2000-5250)/FB Inputs/Value Channel 14 <-> Data Pointer/RawPositionValues[13]
//     Term 27 (AT2000-0250)/Term 28 (AT2000-5250)/FB Inputs/Value Channel 15 <-> Data Pointer/RawPositionValues[14]
//     Term 27 (AT2000-0250)/Term 28 (AT2000-5250)/FB Inputs/Value Channel 16 <-> Data Pointer/RawPositionValues[15]
//     Term 27 (AT2000-0250)/Term 28 (AT2000-5250)/FB Inputs/Value Channel 17 <-> Data Pointer/RawPositionValues[16]
//     Term 27 (AT2000-0250)/Term 28 (AT2000-5250)/FB Inputs/Value Channel 18 <-> Data Pointer/RawPositionValues[17]
//     Term 27 (AT2000-0250)/Term 28 (AT2000-5250)/FB Inputs/Value Channel 19 <-> Data Pointer/RawPositionValues[18]
//     Term 27 (AT2000-0250)/Term 28 (AT2000-5250)/FB Inputs/Value Channel 20 <-> Data Pointer/RawPositionValues[19]
//     Term 27 (AT2000-0250)/Term 28 (AT2000-5250)/FB Inputs/Value Channel 21 <-> Data Pointer/RawPositionValues[20]
//     Term 27 (AT2000-0250)/Term 28 (AT2000-5250)/FB Inputs/Value Channel 22 <-> Data Pointer/RawPositionValues[21]
//     Term 27 (AT2000-0250)/Term 28 (AT2000-5250)/FB Inputs/Value Channel 23 <-> Data Pointer/RawPositionValues[22]
//     Term 27 (AT2000-0250)/Term 28 (AT2000-5250)/FB Inputs/Value Channel 24 <-> Data Pointer/RawPositionValues[23]
//     Term 27 (AT2000-0250)/Term 28 (AT2000-5250)/FB Inputs/Value Channel 25 <-> Data Pointer/RawPositionValues[24]
//     Term 27 (AT2000-0250)/Term 28 (AT2000-5250)/FB Inputs/Value Channel 26 <-> Data Pointer/RawPositionValues[25]
//     Term 27 (AT2000-0250)/Term 28 (AT2000-5250)/FB Inputs/Value Channel 27 <-> Data Pointer/RawPositionValues[26]
//     Term 27 (AT2000-0250)/Term 28 (AT2000-5250)/FB Inputs/Value Channel 28 <-> Data Pointer/RawPositionValues[27]
//     Term 27 (AT2000-0250)/Term 28 (AT2000-5250)/FB Inputs/Value Channel 29 <-> Data Pointer/RawPositionValues[28]
//     Term 27 (AT2000-0250)/Term 28 (AT2000-5250)/FB Inputs/Value Channel 30 <-> Data Pointer/RawPositionValues[29]
//     Term 27 (AT2000-0250)/Term 28 (AT2000-5250)/FB Inputs/Value Channel 31 <-> Data Pointer/RawPositionValues[30]
//     Term 27 (AT2000-0250)/Term 28 (AT2000-5250)/FB Inputs/Value Channel 32 <-> Data Pointer/RawPositionValues[31]
//   Device 17 <-> TcCOM Objects/XTS ProcessingUnit 1/Part 1/Module 15
//     Term 29 (AT2000-0250)/CC Inputs/Current actual value Ch.1 <-> Data Pointer/CurrentActualValues[0]
//     Term 29 (AT2000-0250)/CC Inputs/Current actual value Ch.10 <-> Data Pointer/CurrentActualValues[9]
//     Term 29 (AT2000-0250)/CC Inputs/Current actual value Ch.11 <-> Data Pointer/CurrentActualValues[10]
//     Term 29 (AT2000-0250)/CC Inputs/Current actual value Ch.12 <-> Data Pointer/CurrentActualValues[11]
//     Term 29 (AT2000-0250)/CC Inputs/Current actual value Ch.13 <-> Data Pointer/CurrentActualValues[12]
//     Term 29 (AT2000-0250)/CC Inputs/Current actual value Ch.14 <-> Data Pointer/CurrentActualValues[13]
//     Term 29 (AT2000-0250)/CC Inputs/Current actual value Ch.15 <-> Data Pointer/CurrentActualValues[14]
//     Term 29 (AT2000-0250)/CC Inputs/Current actual value Ch.2 <-> Data Pointer/CurrentActualValues[1]
//     Term 29 (AT2000-0250)/CC Inputs/Current actual value Ch.3 <-> Data Pointer/CurrentActualValues[2]
//     Term 29 (AT2000-0250)/CC Inputs/Current actual value Ch.4 <-> Data Pointer/CurrentActualValues[3]
//     Term 29 (AT2000-0250)/CC Inputs/Current actual value Ch.5 <-> Data Pointer/CurrentActualValues[4]
//     Term 29 (AT2000-0250)/CC Inputs/Current actual value Ch.6 <-> Data Pointer/CurrentActualValues[5]
//     Term 29 (AT2000-0250)/CC Inputs/Current actual value Ch.7 <-> Data Pointer/CurrentActualValues[6]
//     Term 29 (AT2000-0250)/CC Inputs/Current actual value Ch.8 <-> Data Pointer/CurrentActualValues[7]
//     Term 29 (AT2000-0250)/CC Inputs/Current actual value Ch.9 <-> Data Pointer/CurrentActualValues[8]
//     Term 29 (AT2000-0250)/CC Inputs/Status <-> Data Pointer/Status
//     Term 29 (AT2000-0250)/CC Outputs/Control <-> Data Pointer/Control
//     Term 29 (AT2000-0250)/CC Outputs/Current setpoint value Ch.1 <-> Data Pointer/CurrentSetpointValues[0]
//     Term 29 (AT2000-0250)/CC Outputs/Current setpoint value Ch.10 <-> Data Pointer/CurrentSetpointValues[9]
//     Term 29 (AT2000-0250)/CC Outputs/Current setpoint value Ch.11 <-> Data Pointer/CurrentSetpointValues[10]
//     Term 29 (AT2000-0250)/CC Outputs/Current setpoint value Ch.12 <-> Data Pointer/CurrentSetpointValues[11]
//     Term 29 (AT2000-0250)/CC Outputs/Current setpoint value Ch.13 <-> Data Pointer/CurrentSetpointValues[12]
//     Term 29 (AT2000-0250)/CC Outputs/Current setpoint value Ch.14 <-> Data Pointer/CurrentSetpointValues[13]
//     Term 29 (AT2000-0250)/CC Outputs/Current setpoint value Ch.15 <-> Data Pointer/CurrentSetpointValues[14]
//     Term 29 (AT2000-0250)/CC Outputs/Current setpoint value Ch.2 <-> Data Pointer/CurrentSetpointValues[1]
//     Term 29 (AT2000-0250)/CC Outputs/Current setpoint value Ch.3 <-> Data Pointer/CurrentSetpointValues[2]
//     Term 29 (AT2000-0250)/CC Outputs/Current setpoint value Ch.4 <-> Data Pointer/CurrentSetpointValues[3]
//     Term 29 (AT2000-0250)/CC Outputs/Current setpoint value Ch.5 <-> Data Pointer/CurrentSetpointValues[4]
//     Term 29 (AT2000-0250)/CC Outputs/Current setpoint value Ch.6 <-> Data Pointer/CurrentSetpointValues[5]
//     Term 29 (AT2000-0250)/CC Outputs/Current setpoint value Ch.7 <-> Data Pointer/CurrentSetpointValues[6]
//     Term 29 (AT2000-0250)/CC Outputs/Current setpoint value Ch.8 <-> Data Pointer/CurrentSetpointValues[7]
//     Term 29 (AT2000-0250)/CC Outputs/Current setpoint value Ch.9 <-> Data Pointer/CurrentSetpointValues[8]
//     Term 29 (AT2000-0250)/Term 30 (AT2000-5250)/FB Inputs/Value Channel 01 <-> Data Pointer/RawPositionValues[0]
//     Term 29 (AT2000-0250)/Term 30 (AT2000-5250)/FB Inputs/Value Channel 02 <-> Data Pointer/RawPositionValues[1]
//     Term 29 (AT2000-0250)/Term 30 (AT2000-5250)/FB Inputs/Value Channel 03 <-> Data Pointer/RawPositionValues[2]
//     Term 29 (AT2000-0250)/Term 30 (AT2000-5250)/FB Inputs/Value Channel 04 <-> Data Pointer/RawPositionValues[3]
//     Term 29 (AT2000-0250)/Term 30 (AT2000-5250)/FB Inputs/Value Channel 05 <-> Data Pointer/RawPositionValues[4]
//     Term 29 (AT2000-0250)/Term 30 (AT2000-5250)/FB Inputs/Value Channel 06 <-> Data Pointer/RawPositionValues[5]
//     Term 29 (AT2000-0250)/Term 30 (AT2000-5250)/FB Inputs/Value Channel 07 <-> Data Pointer/RawPositionValues[6]
//     Term 29 (AT2000-0250)/Term 30 (AT2000-5250)/FB Inputs/Value Channel 08 <-> Data Pointer/RawPositionValues[7]
//     Term 29 (AT2000-0250)/Term 30 (AT2000-5250)/FB Inputs/Value Channel 09 <-> Data Pointer/RawPositionValues[8]
//     Term 29 (AT2000-0250)/Term 30 (AT2000-5250)/FB Inputs/Value Channel 10 <-> Data Pointer/RawPositionValues[9]
//     Term 29 (AT2000-0250)/Term 30 (AT2000-5250)/FB Inputs/Value Channel 11 <-> Data Pointer/RawPositionValues[10]
//     Term 29 (AT2000-0250)/Term 30 (AT2000-5250)/FB Inputs/Value Channel 12 <-> Data Pointer/RawPositionValues[11]
//     Term 29 (AT2000-0250)/Term 30 (AT2000-5250)/FB Inputs/Value Channel 13 <-> Data Pointer/RawPositionValues[12]
//     Term 29 (AT2000-0250)/Term 30 (AT2000-5250)/FB Inputs/Value Channel 14 <-> Data Pointer/RawPositionValues[13]
//     Term 29 (AT2000-0250)/Term 30 (AT2000-5250)/FB Inputs/Value Channel 15 <-> Data Pointer/RawPositionValues[14]
//     Term 29 (AT2000-0250)/Term 30 (AT2000-5250)/FB Inputs/Value Channel 16 <-> Data Pointer/RawPositionValues[15]
//     Term 29 (AT2000-0250)/Term 30 (AT2000-5250)/FB Inputs/Value Channel 17 <-> Data Pointer/RawPositionValues[16]
//     Term 29 (AT2000-0250)/Term 30 (AT2000-5250)/FB Inputs/Value Channel 18 <-> Data Pointer/RawPositionValues[17]
//     Term 29 (AT2000-0250)/Term 30 (AT2000-5250)/FB Inputs/Value Channel 19 <-> Data Pointer/RawPositionValues[18]
//     Term 29 (AT2000-0250)/Term 30 (AT2000-5250)/FB Inputs/Value Channel 20 <-> Data Pointer/RawPositionValues[19]
//     Term 29 (AT2000-0250)/Term 30 (AT2000-5250)/FB Inputs/Value Channel 21 <-> Data Pointer/RawPositionValues[20]
//     Term 29 (AT2000-0250)/Term 30 (AT2000-5250)/FB Inputs/Value Channel 22 <-> Data Pointer/RawPositionValues[21]
//     Term 29 (AT2000-0250)/Term 30 (AT2000-5250)/FB Inputs/Value Channel 23 <-> Data Pointer/RawPositionValues[22]
//     Term 29 (AT2000-0250)/Term 30 (AT2000-5250)/FB Inputs/Value Channel 24 <-> Data Pointer/RawPositionValues[23]
//     Term 29 (AT2000-0250)/Term 30 (AT2000-5250)/FB Inputs/Value Channel 25 <-> Data Pointer/RawPositionValues[24]
//     Term 29 (AT2000-0250)/Term 30 (AT2000-5250)/FB Inputs/Value Channel 26 <-> Data Pointer/RawPositionValues[25]
//     Term 29 (AT2000-0250)/Term 30 (AT2000-5250)/FB Inputs/Value Channel 27 <-> Data Pointer/RawPositionValues[26]
//     Term 29 (AT2000-0250)/Term 30 (AT2000-5250)/FB Inputs/Value Channel 28 <-> Data Pointer/RawPositionValues[27]
//     Term 29 (AT2000-0250)/Term 30 (AT2000-5250)/FB Inputs/Value Channel 29 <-> Data Pointer/RawPositionValues[28]
//     Term 29 (AT2000-0250)/Term 30 (AT2000-5250)/FB Inputs/Value Channel 30 <-> Data Pointer/RawPositionValues[29]
//     Term 29 (AT2000-0250)/Term 30 (AT2000-5250)/FB Inputs/Value Channel 31 <-> Data Pointer/RawPositionValues[30]
//     Term 29 (AT2000-0250)/Term 30 (AT2000-5250)/FB Inputs/Value Channel 32 <-> Data Pointer/RawPositionValues[31]
//   Device 17 <-> TcCOM Objects/XTS ProcessingUnit 1/Part 1/Module 16
//     Term 31 (AT2000-0250)/CC Inputs/Current actual value Ch.1 <-> Data Pointer/CurrentActualValues[0]
//     Term 31 (AT2000-0250)/CC Inputs/Current actual value Ch.10 <-> Data Pointer/CurrentActualValues[9]
//     Term 31 (AT2000-0250)/CC Inputs/Current actual value Ch.11 <-> Data Pointer/CurrentActualValues[10]
//     Term 31 (AT2000-0250)/CC Inputs/Current actual value Ch.12 <-> Data Pointer/CurrentActualValues[11]
//     Term 31 (AT2000-0250)/CC Inputs/Current actual value Ch.13 <-> Data Pointer/CurrentActualValues[12]
//     Term 31 (AT2000-0250)/CC Inputs/Current actual value Ch.14 <-> Data Pointer/CurrentActualValues[13]
//     Term 31 (AT2000-0250)/CC Inputs/Current actual value Ch.15 <-> Data Pointer/CurrentActualValues[14]
//     Term 31 (AT2000-0250)/CC Inputs/Current actual value Ch.2 <-> Data Pointer/CurrentActualValues[1]
//     Term 31 (AT2000-0250)/CC Inputs/Current actual value Ch.3 <-> Data Pointer/CurrentActualValues[2]
//     Term 31 (AT2000-0250)/CC Inputs/Current actual value Ch.4 <-> Data Pointer/CurrentActualValues[3]
//     Term 31 (AT2000-0250)/CC Inputs/Current actual value Ch.5 <-> Data Pointer/CurrentActualValues[4]
//     Term 31 (AT2000-0250)/CC Inputs/Current actual value Ch.6 <-> Data Pointer/CurrentActualValues[5]
//     Term 31 (AT2000-0250)/CC Inputs/Current actual value Ch.7 <-> Data Pointer/CurrentActualValues[6]
//     Term 31 (AT2000-0250)/CC Inputs/Current actual value Ch.8 <-> Data Pointer/CurrentActualValues[7]
//     Term 31 (AT2000-0250)/CC Inputs/Current actual value Ch.9 <-> Data Pointer/CurrentActualValues[8]
//     Term 31 (AT2000-0250)/CC Inputs/Status <-> Data Pointer/Status
//     Term 31 (AT2000-0250)/CC Outputs/Control <-> Data Pointer/Control
//     Term 31 (AT2000-0250)/CC Outputs/Current setpoint value Ch.1 <-> Data Pointer/CurrentSetpointValues[0]
//     Term 31 (AT2000-0250)/CC Outputs/Current setpoint value Ch.10 <-> Data Pointer/CurrentSetpointValues[9]
//     Term 31 (AT2000-0250)/CC Outputs/Current setpoint value Ch.11 <-> Data Pointer/CurrentSetpointValues[10]
//     Term 31 (AT2000-0250)/CC Outputs/Current setpoint value Ch.12 <-> Data Pointer/CurrentSetpointValues[11]
//     Term 31 (AT2000-0250)/CC Outputs/Current setpoint value Ch.13 <-> Data Pointer/CurrentSetpointValues[12]
//     Term 31 (AT2000-0250)/CC Outputs/Current setpoint value Ch.14 <-> Data Pointer/CurrentSetpointValues[13]
//     Term 31 (AT2000-0250)/CC Outputs/Current setpoint value Ch.15 <-> Data Pointer/CurrentSetpointValues[14]
//     Term 31 (AT2000-0250)/CC Outputs/Current setpoint value Ch.2 <-> Data Pointer/CurrentSetpointValues[1]
//     Term 31 (AT2000-0250)/CC Outputs/Current setpoint value Ch.3 <-> Data Pointer/CurrentSetpointValues[2]
//     Term 31 (AT2000-0250)/CC Outputs/Current setpoint value Ch.4 <-> Data Pointer/CurrentSetpointValues[3]
//     Term 31 (AT2000-0250)/CC Outputs/Current setpoint value Ch.5 <-> Data Pointer/CurrentSetpointValues[4]
//     Term 31 (AT2000-0250)/CC Outputs/Current setpoint value Ch.6 <-> Data Pointer/CurrentSetpointValues[5]
//     Term 31 (AT2000-0250)/CC Outputs/Current setpoint value Ch.7 <-> Data Pointer/CurrentSetpointValues[6]
//     Term 31 (AT2000-0250)/CC Outputs/Current setpoint value Ch.8 <-> Data Pointer/CurrentSetpointValues[7]
//     Term 31 (AT2000-0250)/CC Outputs/Current setpoint value Ch.9 <-> Data Pointer/CurrentSetpointValues[8]
//     Term 31 (AT2000-0250)/Term 32 (AT2000-5250)/FB Inputs/Value Channel 01 <-> Data Pointer/RawPositionValues[0]
//     Term 31 (AT2000-0250)/Term 32 (AT2000-5250)/FB Inputs/Value Channel 02 <-> Data Pointer/RawPositionValues[1]
//     Term 31 (AT2000-0250)/Term 32 (AT2000-5250)/FB Inputs/Value Channel 03 <-> Data Pointer/RawPositionValues[2]
//     Term 31 (AT2000-0250)/Term 32 (AT2000-5250)/FB Inputs/Value Channel 04 <-> Data Pointer/RawPositionValues[3]
//     Term 31 (AT2000-0250)/Term 32 (AT2000-5250)/FB Inputs/Value Channel 05 <-> Data Pointer/RawPositionValues[4]
//     Term 31 (AT2000-0250)/Term 32 (AT2000-5250)/FB Inputs/Value Channel 06 <-> Data Pointer/RawPositionValues[5]
//     Term 31 (AT2000-0250)/Term 32 (AT2000-5250)/FB Inputs/Value Channel 07 <-> Data Pointer/RawPositionValues[6]
//     Term 31 (AT2000-0250)/Term 32 (AT2000-5250)/FB Inputs/Value Channel 08 <-> Data Pointer/RawPositionValues[7]
//     Term 31 (AT2000-0250)/Term 32 (AT2000-5250)/FB Inputs/Value Channel 09 <-> Data Pointer/RawPositionValues[8]
//     Term 31 (AT2000-0250)/Term 32 (AT2000-5250)/FB Inputs/Value Channel 10 <-> Data Pointer/RawPositionValues[9]
//     Term 31 (AT2000-0250)/Term 32 (AT2000-5250)/FB Inputs/Value Channel 11 <-> Data Pointer/RawPositionValues[10]
//     Term 31 (AT2000-0250)/Term 32 (AT2000-5250)/FB Inputs/Value Channel 12 <-> Data Pointer/RawPositionValues[11]
//     Term 31 (AT2000-0250)/Term 32 (AT2000-5250)/FB Inputs/Value Channel 13 <-> Data Pointer/RawPositionValues[12]
//     Term 31 (AT2000-0250)/Term 32 (AT2000-5250)/FB Inputs/Value Channel 14 <-> Data Pointer/RawPositionValues[13]
//     Term 31 (AT2000-0250)/Term 32 (AT2000-5250)/FB Inputs/Value Channel 15 <-> Data Pointer/RawPositionValues[14]
//     Term 31 (AT2000-0250)/Term 32 (AT2000-5250)/FB Inputs/Value Channel 16 <-> Data Pointer/RawPositionValues[15]
//     Term 31 (AT2000-0250)/Term 32 (AT2000-5250)/FB Inputs/Value Channel 17 <-> Data Pointer/RawPositionValues[16]
//     Term 31 (AT2000-0250)/Term 32 (AT2000-5250)/FB Inputs/Value Channel 18 <-> Data Pointer/RawPositionValues[17]
//     Term 31 (AT2000-0250)/Term 32 (AT2000-5250)/FB Inputs/Value Channel 19 <-> Data Pointer/RawPositionValues[18]
//     Term 31 (AT2000-0250)/Term 32 (AT2000-5250)/FB Inputs/Value Channel 20 <-> Data Pointer/RawPositionValues[19]
//     Term 31 (AT2000-0250)/Term 32 (AT2000-5250)/FB Inputs/Value Channel 21 <-> Data Pointer/RawPositionValues[20]
//     Term 31 (AT2000-0250)/Term 32 (AT2000-5250)/FB Inputs/Value Channel 22 <-> Data Pointer/RawPositionValues[21]
//     Term 31 (AT2000-0250)/Term 32 (AT2000-5250)/FB Inputs/Value Channel 23 <-> Data Pointer/RawPositionValues[22]
//     Term 31 (AT2000-0250)/Term 32 (AT2000-5250)/FB Inputs/Value Channel 24 <-> Data Pointer/RawPositionValues[23]
//     Term 31 (AT2000-0250)/Term 32 (AT2000-5250)/FB Inputs/Value Channel 25 <-> Data Pointer/RawPositionValues[24]
//     Term 31 (AT2000-0250)/Term 32 (AT2000-5250)/FB Inputs/Value Channel 26 <-> Data Pointer/RawPositionValues[25]
//     Term 31 (AT2000-0250)/Term 32 (AT2000-5250)/FB Inputs/Value Channel 27 <-> Data Pointer/RawPositionValues[26]
//     Term 31 (AT2000-0250)/Term 32 (AT2000-5250)/FB Inputs/Value Channel 28 <-> Data Pointer/RawPositionValues[27]
//     Term 31 (AT2000-0250)/Term 32 (AT2000-5250)/FB Inputs/Value Channel 29 <-> Data Pointer/RawPositionValues[28]
//     Term 31 (AT2000-0250)/Term 32 (AT2000-5250)/FB Inputs/Value Channel 30 <-> Data Pointer/RawPositionValues[29]
//     Term 31 (AT2000-0250)/Term 32 (AT2000-5250)/FB Inputs/Value Channel 31 <-> Data Pointer/RawPositionValues[30]
//     Term 31 (AT2000-0250)/Term 32 (AT2000-5250)/FB Inputs/Value Channel 32 <-> Data Pointer/RawPositionValues[31]
//   Device 17 <-> TcCOM Objects/XTS ProcessingUnit 1/Part 1/Module 17
//     Term 33 (AT2000-0250)/CC Inputs/Current actual value Ch.1 <-> Data Pointer/CurrentActualValues[0]
//     Term 33 (AT2000-0250)/CC Inputs/Current actual value Ch.10 <-> Data Pointer/CurrentActualValues[9]
//     Term 33 (AT2000-0250)/CC Inputs/Current actual value Ch.11 <-> Data Pointer/CurrentActualValues[10]
//     Term 33 (AT2000-0250)/CC Inputs/Current actual value Ch.12 <-> Data Pointer/CurrentActualValues[11]
//     Term 33 (AT2000-0250)/CC Inputs/Current actual value Ch.13 <-> Data Pointer/CurrentActualValues[12]
//     Term 33 (AT2000-0250)/CC Inputs/Current actual value Ch.14 <-> Data Pointer/CurrentActualValues[13]
//     Term 33 (AT2000-0250)/CC Inputs/Current actual value Ch.15 <-> Data Pointer/CurrentActualValues[14]
//     Term 33 (AT2000-0250)/CC Inputs/Current actual value Ch.2 <-> Data Pointer/CurrentActualValues[1]
//     Term 33 (AT2000-0250)/CC Inputs/Current actual value Ch.3 <-> Data Pointer/CurrentActualValues[2]
//     Term 33 (AT2000-0250)/CC Inputs/Current actual value Ch.4 <-> Data Pointer/CurrentActualValues[3]
//     Term 33 (AT2000-0250)/CC Inputs/Current actual value Ch.5 <-> Data Pointer/CurrentActualValues[4]
//     Term 33 (AT2000-0250)/CC Inputs/Current actual value Ch.6 <-> Data Pointer/CurrentActualValues[5]
//     Term 33 (AT2000-0250)/CC Inputs/Current actual value Ch.7 <-> Data Pointer/CurrentActualValues[6]
//     Term 33 (AT2000-0250)/CC Inputs/Current actual value Ch.8 <-> Data Pointer/CurrentActualValues[7]
//     Term 33 (AT2000-0250)/CC Inputs/Current actual value Ch.9 <-> Data Pointer/CurrentActualValues[8]
//     Term 33 (AT2000-0250)/CC Inputs/Status <-> Data Pointer/Status
//     Term 33 (AT2000-0250)/CC Outputs/Control <-> Data Pointer/Control
//     Term 33 (AT2000-0250)/CC Outputs/Current setpoint value Ch.1 <-> Data Pointer/CurrentSetpointValues[0]
//     Term 33 (AT2000-0250)/CC Outputs/Current setpoint value Ch.10 <-> Data Pointer/CurrentSetpointValues[9]
//     Term 33 (AT2000-0250)/CC Outputs/Current setpoint value Ch.11 <-> Data Pointer/CurrentSetpointValues[10]
//     Term 33 (AT2000-0250)/CC Outputs/Current setpoint value Ch.12 <-> Data Pointer/CurrentSetpointValues[11]
//     Term 33 (AT2000-0250)/CC Outputs/Current setpoint value Ch.13 <-> Data Pointer/CurrentSetpointValues[12]
//     Term 33 (AT2000-0250)/CC Outputs/Current setpoint value Ch.14 <-> Data Pointer/CurrentSetpointValues[13]
//     Term 33 (AT2000-0250)/CC Outputs/Current setpoint value Ch.15 <-> Data Pointer/CurrentSetpointValues[14]
//     Term 33 (AT2000-0250)/CC Outputs/Current setpoint value Ch.2 <-> Data Pointer/CurrentSetpointValues[1]
//     Term 33 (AT2000-0250)/CC Outputs/Current setpoint value Ch.3 <-> Data Pointer/CurrentSetpointValues[2]
//     Term 33 (AT2000-0250)/CC Outputs/Current setpoint value Ch.4 <-> Data Pointer/CurrentSetpointValues[3]
//     Term 33 (AT2000-0250)/CC Outputs/Current setpoint value Ch.5 <-> Data Pointer/CurrentSetpointValues[4]
//     Term 33 (AT2000-0250)/CC Outputs/Current setpoint value Ch.6 <-> Data Pointer/CurrentSetpointValues[5]
//     Term 33 (AT2000-0250)/CC Outputs/Current setpoint value Ch.7 <-> Data Pointer/CurrentSetpointValues[6]
//     Term 33 (AT2000-0250)/CC Outputs/Current setpoint value Ch.8 <-> Data Pointer/CurrentSetpointValues[7]
//     Term 33 (AT2000-0250)/CC Outputs/Current setpoint value Ch.9 <-> Data Pointer/CurrentSetpointValues[8]
//     Term 33 (AT2000-0250)/Term 34 (AT2000-5250)/FB Inputs/Value Channel 01 <-> Data Pointer/RawPositionValues[0]
//     Term 33 (AT2000-0250)/Term 34 (AT2000-5250)/FB Inputs/Value Channel 02 <-> Data Pointer/RawPositionValues[1]
//     Term 33 (AT2000-0250)/Term 34 (AT2000-5250)/FB Inputs/Value Channel 03 <-> Data Pointer/RawPositionValues[2]
//     Term 33 (AT2000-0250)/Term 34 (AT2000-5250)/FB Inputs/Value Channel 04 <-> Data Pointer/RawPositionValues[3]
//     Term 33 (AT2000-0250)/Term 34 (AT2000-5250)/FB Inputs/Value Channel 05 <-> Data Pointer/RawPositionValues[4]
//     Term 33 (AT2000-0250)/Term 34 (AT2000-5250)/FB Inputs/Value Channel 06 <-> Data Pointer/RawPositionValues[5]
//     Term 33 (AT2000-0250)/Term 34 (AT2000-5250)/FB Inputs/Value Channel 07 <-> Data Pointer/RawPositionValues[6]
//     Term 33 (AT2000-0250)/Term 34 (AT2000-5250)/FB Inputs/Value Channel 08 <-> Data Pointer/RawPositionValues[7]
//     Term 33 (AT2000-0250)/Term 34 (AT2000-5250)/FB Inputs/Value Channel 09 <-> Data Pointer/RawPositionValues[8]
//     Term 33 (AT2000-0250)/Term 34 (AT2000-5250)/FB Inputs/Value Channel 10 <-> Data Pointer/RawPositionValues[9]
//     Term 33 (AT2000-0250)/Term 34 (AT2000-5250)/FB Inputs/Value Channel 11 <-> Data Pointer/RawPositionValues[10]
//     Term 33 (AT2000-0250)/Term 34 (AT2000-5250)/FB Inputs/Value Channel 12 <-> Data Pointer/RawPositionValues[11]
//     Term 33 (AT2000-0250)/Term 34 (AT2000-5250)/FB Inputs/Value Channel 13 <-> Data Pointer/RawPositionValues[12]
//     Term 33 (AT2000-0250)/Term 34 (AT2000-5250)/FB Inputs/Value Channel 14 <-> Data Pointer/RawPositionValues[13]
//     Term 33 (AT2000-0250)/Term 34 (AT2000-5250)/FB Inputs/Value Channel 15 <-> Data Pointer/RawPositionValues[14]
//     Term 33 (AT2000-0250)/Term 34 (AT2000-5250)/FB Inputs/Value Channel 16 <-> Data Pointer/RawPositionValues[15]
//     Term 33 (AT2000-0250)/Term 34 (AT2000-5250)/FB Inputs/Value Channel 17 <-> Data Pointer/RawPositionValues[16]
//     Term 33 (AT2000-0250)/Term 34 (AT2000-5250)/FB Inputs/Value Channel 18 <-> Data Pointer/RawPositionValues[17]
//     Term 33 (AT2000-0250)/Term 34 (AT2000-5250)/FB Inputs/Value Channel 19 <-> Data Pointer/RawPositionValues[18]
//     Term 33 (AT2000-0250)/Term 34 (AT2000-5250)/FB Inputs/Value Channel 20 <-> Data Pointer/RawPositionValues[19]
//     Term 33 (AT2000-0250)/Term 34 (AT2000-5250)/FB Inputs/Value Channel 21 <-> Data Pointer/RawPositionValues[20]
//     Term 33 (AT2000-0250)/Term 34 (AT2000-5250)/FB Inputs/Value Channel 22 <-> Data Pointer/RawPositionValues[21]
//     Term 33 (AT2000-0250)/Term 34 (AT2000-5250)/FB Inputs/Value Channel 23 <-> Data Pointer/RawPositionValues[22]
//     Term 33 (AT2000-0250)/Term 34 (AT2000-5250)/FB Inputs/Value Channel 24 <-> Data Pointer/RawPositionValues[23]
//     Term 33 (AT2000-0250)/Term 34 (AT2000-5250)/FB Inputs/Value Channel 25 <-> Data Pointer/RawPositionValues[24]
//     Term 33 (AT2000-0250)/Term 34 (AT2000-5250)/FB Inputs/Value Channel 26 <-> Data Pointer/RawPositionValues[25]
//     Term 33 (AT2000-0250)/Term 34 (AT2000-5250)/FB Inputs/Value Channel 27 <-> Data Pointer/RawPositionValues[26]
//     Term 33 (AT2000-0250)/Term 34 (AT2000-5250)/FB Inputs/Value Channel 28 <-> Data Pointer/RawPositionValues[27]
//     Term 33 (AT2000-0250)/Term 34 (AT2000-5250)/FB Inputs/Value Channel 29 <-> Data Pointer/RawPositionValues[28]
//     Term 33 (AT2000-0250)/Term 34 (AT2000-5250)/FB Inputs/Value Channel 30 <-> Data Pointer/RawPositionValues[29]
//     Term 33 (AT2000-0250)/Term 34 (AT2000-5250)/FB Inputs/Value Channel 31 <-> Data Pointer/RawPositionValues[30]
//     Term 33 (AT2000-0250)/Term 34 (AT2000-5250)/FB Inputs/Value Channel 32 <-> Data Pointer/RawPositionValues[31]
//   Device 17 <-> TcCOM Objects/XTS ProcessingUnit 1/Part 1/Module 18
//     Term 35 (AT2000-0250)/CC Inputs/Current actual value Ch.1 <-> Data Pointer/CurrentActualValues[0]
//     Term 35 (AT2000-0250)/CC Inputs/Current actual value Ch.10 <-> Data Pointer/CurrentActualValues[9]
//     Term 35 (AT2000-0250)/CC Inputs/Current actual value Ch.11 <-> Data Pointer/CurrentActualValues[10]
//     Term 35 (AT2000-0250)/CC Inputs/Current actual value Ch.12 <-> Data Pointer/CurrentActualValues[11]
//     Term 35 (AT2000-0250)/CC Inputs/Current actual value Ch.13 <-> Data Pointer/CurrentActualValues[12]
//     Term 35 (AT2000-0250)/CC Inputs/Current actual value Ch.14 <-> Data Pointer/CurrentActualValues[13]
//     Term 35 (AT2000-0250)/CC Inputs/Current actual value Ch.15 <-> Data Pointer/CurrentActualValues[14]
//     Term 35 (AT2000-0250)/CC Inputs/Current actual value Ch.2 <-> Data Pointer/CurrentActualValues[1]
//     Term 35 (AT2000-0250)/CC Inputs/Current actual value Ch.3 <-> Data Pointer/CurrentActualValues[2]
//     Term 35 (AT2000-0250)/CC Inputs/Current actual value Ch.4 <-> Data Pointer/CurrentActualValues[3]
//     Term 35 (AT2000-0250)/CC Inputs/Current actual value Ch.5 <-> Data Pointer/CurrentActualValues[4]
//     Term 35 (AT2000-0250)/CC Inputs/Current actual value Ch.6 <-> Data Pointer/CurrentActualValues[5]
//     Term 35 (AT2000-0250)/CC Inputs/Current actual value Ch.7 <-> Data Pointer/CurrentActualValues[6]
//     Term 35 (AT2000-0250)/CC Inputs/Current actual value Ch.8 <-> Data Pointer/CurrentActualValues[7]
//     Term 35 (AT2000-0250)/CC Inputs/Current actual value Ch.9 <-> Data Pointer/CurrentActualValues[8]
//     Term 35 (AT2000-0250)/CC Inputs/Status <-> Data Pointer/Status
//     Term 35 (AT2000-0250)/CC Outputs/Control <-> Data Pointer/Control
//     Term 35 (AT2000-0250)/CC Outputs/Current setpoint value Ch.1 <-> Data Pointer/CurrentSetpointValues[0]
//     Term 35 (AT2000-0250)/CC Outputs/Current setpoint value Ch.10 <-> Data Pointer/CurrentSetpointValues[9]
//     Term 35 (AT2000-0250)/CC Outputs/Current setpoint value Ch.11 <-> Data Pointer/CurrentSetpointValues[10]
//     Term 35 (AT2000-0250)/CC Outputs/Current setpoint value Ch.12 <-> Data Pointer/CurrentSetpointValues[11]
//     Term 35 (AT2000-0250)/CC Outputs/Current setpoint value Ch.13 <-> Data Pointer/CurrentSetpointValues[12]
//     Term 35 (AT2000-0250)/CC Outputs/Current setpoint value Ch.14 <-> Data Pointer/CurrentSetpointValues[13]
//     Term 35 (AT2000-0250)/CC Outputs/Current setpoint value Ch.15 <-> Data Pointer/CurrentSetpointValues[14]
//     Term 35 (AT2000-0250)/CC Outputs/Current setpoint value Ch.2 <-> Data Pointer/CurrentSetpointValues[1]
//     Term 35 (AT2000-0250)/CC Outputs/Current setpoint value Ch.3 <-> Data Pointer/CurrentSetpointValues[2]
//     Term 35 (AT2000-0250)/CC Outputs/Current setpoint value Ch.4 <-> Data Pointer/CurrentSetpointValues[3]
//     Term 35 (AT2000-0250)/CC Outputs/Current setpoint value Ch.5 <-> Data Pointer/CurrentSetpointValues[4]
//     Term 35 (AT2000-0250)/CC Outputs/Current setpoint value Ch.6 <-> Data Pointer/CurrentSetpointValues[5]
//     Term 35 (AT2000-0250)/CC Outputs/Current setpoint value Ch.7 <-> Data Pointer/CurrentSetpointValues[6]
//     Term 35 (AT2000-0250)/CC Outputs/Current setpoint value Ch.8 <-> Data Pointer/CurrentSetpointValues[7]
//     Term 35 (AT2000-0250)/CC Outputs/Current setpoint value Ch.9 <-> Data Pointer/CurrentSetpointValues[8]
//     Term 35 (AT2000-0250)/Term 36 (AT2000-5250)/FB Inputs/Value Channel 01 <-> Data Pointer/RawPositionValues[0]
//     Term 35 (AT2000-0250)/Term 36 (AT2000-5250)/FB Inputs/Value Channel 02 <-> Data Pointer/RawPositionValues[1]
//     Term 35 (AT2000-0250)/Term 36 (AT2000-5250)/FB Inputs/Value Channel 03 <-> Data Pointer/RawPositionValues[2]
//     Term 35 (AT2000-0250)/Term 36 (AT2000-5250)/FB Inputs/Value Channel 04 <-> Data Pointer/RawPositionValues[3]
//     Term 35 (AT2000-0250)/Term 36 (AT2000-5250)/FB Inputs/Value Channel 05 <-> Data Pointer/RawPositionValues[4]
//     Term 35 (AT2000-0250)/Term 36 (AT2000-5250)/FB Inputs/Value Channel 06 <-> Data Pointer/RawPositionValues[5]
//     Term 35 (AT2000-0250)/Term 36 (AT2000-5250)/FB Inputs/Value Channel 07 <-> Data Pointer/RawPositionValues[6]
//     Term 35 (AT2000-0250)/Term 36 (AT2000-5250)/FB Inputs/Value Channel 08 <-> Data Pointer/RawPositionValues[7]
//     Term 35 (AT2000-0250)/Term 36 (AT2000-5250)/FB Inputs/Value Channel 09 <-> Data Pointer/RawPositionValues[8]
//     Term 35 (AT2000-0250)/Term 36 (AT2000-5250)/FB Inputs/Value Channel 10 <-> Data Pointer/RawPositionValues[9]
//     Term 35 (AT2000-0250)/Term 36 (AT2000-5250)/FB Inputs/Value Channel 11 <-> Data Pointer/RawPositionValues[10]
//     Term 35 (AT2000-0250)/Term 36 (AT2000-5250)/FB Inputs/Value Channel 12 <-> Data Pointer/RawPositionValues[11]
//     Term 35 (AT2000-0250)/Term 36 (AT2000-5250)/FB Inputs/Value Channel 13 <-> Data Pointer/RawPositionValues[12]
//     Term 35 (AT2000-0250)/Term 36 (AT2000-5250)/FB Inputs/Value Channel 14 <-> Data Pointer/RawPositionValues[13]
//     Term 35 (AT2000-0250)/Term 36 (AT2000-5250)/FB Inputs/Value Channel 15 <-> Data Pointer/RawPositionValues[14]
//     Term 35 (AT2000-0250)/Term 36 (AT2000-5250)/FB Inputs/Value Channel 16 <-> Data Pointer/RawPositionValues[15]
//     Term 35 (AT2000-0250)/Term 36 (AT2000-5250)/FB Inputs/Value Channel 17 <-> Data Pointer/RawPositionValues[16]
//     Term 35 (AT2000-0250)/Term 36 (AT2000-5250)/FB Inputs/Value Channel 18 <-> Data Pointer/RawPositionValues[17]
//     Term 35 (AT2000-0250)/Term 36 (AT2000-5250)/FB Inputs/Value Channel 19 <-> Data Pointer/RawPositionValues[18]
//     Term 35 (AT2000-0250)/Term 36 (AT2000-5250)/FB Inputs/Value Channel 20 <-> Data Pointer/RawPositionValues[19]
//     Term 35 (AT2000-0250)/Term 36 (AT2000-5250)/FB Inputs/Value Channel 21 <-> Data Pointer/RawPositionValues[20]
//     Term 35 (AT2000-0250)/Term 36 (AT2000-5250)/FB Inputs/Value Channel 22 <-> Data Pointer/RawPositionValues[21]
//     Term 35 (AT2000-0250)/Term 36 (AT2000-5250)/FB Inputs/Value Channel 23 <-> Data Pointer/RawPositionValues[22]
//     Term 35 (AT2000-0250)/Term 36 (AT2000-5250)/FB Inputs/Value Channel 24 <-> Data Pointer/RawPositionValues[23]
//     Term 35 (AT2000-0250)/Term 36 (AT2000-5250)/FB Inputs/Value Channel 25 <-> Data Pointer/RawPositionValues[24]
//     Term 35 (AT2000-0250)/Term 36 (AT2000-5250)/FB Inputs/Value Channel 26 <-> Data Pointer/RawPositionValues[25]
//     Term 35 (AT2000-0250)/Term 36 (AT2000-5250)/FB Inputs/Value Channel 27 <-> Data Pointer/RawPositionValues[26]
//     Term 35 (AT2000-0250)/Term 36 (AT2000-5250)/FB Inputs/Value Channel 28 <-> Data Pointer/RawPositionValues[27]
//     Term 35 (AT2000-0250)/Term 36 (AT2000-5250)/FB Inputs/Value Channel 29 <-> Data Pointer/RawPositionValues[28]
//     Term 35 (AT2000-0250)/Term 36 (AT2000-5250)/FB Inputs/Value Channel 30 <-> Data Pointer/RawPositionValues[29]
//     Term 35 (AT2000-0250)/Term 36 (AT2000-5250)/FB Inputs/Value Channel 31 <-> Data Pointer/RawPositionValues[30]
//     Term 35 (AT2000-0250)/Term 36 (AT2000-5250)/FB Inputs/Value Channel 32 <-> Data Pointer/RawPositionValues[31]
//   Device 18 <-> TcCOM Objects/XTS ProcessingUnit 1/Part 1/Module 19
//     Term 37 (AT2002-0250)/CC Inputs/Current actual value Ch.1 <-> Data Pointer/CurrentActualValues[0]
//     Term 37 (AT2002-0250)/CC Inputs/Current actual value Ch.10 <-> Data Pointer/CurrentActualValues[9]
//     Term 37 (AT2002-0250)/CC Inputs/Current actual value Ch.11 <-> Data Pointer/CurrentActualValues[10]
//     Term 37 (AT2002-0250)/CC Inputs/Current actual value Ch.12 <-> Data Pointer/CurrentActualValues[11]
//     Term 37 (AT2002-0250)/CC Inputs/Current actual value Ch.13 <-> Data Pointer/CurrentActualValues[12]
//     Term 37 (AT2002-0250)/CC Inputs/Current actual value Ch.14 <-> Data Pointer/CurrentActualValues[13]
//     Term 37 (AT2002-0250)/CC Inputs/Current actual value Ch.15 <-> Data Pointer/CurrentActualValues[14]
//     Term 37 (AT2002-0250)/CC Inputs/Current actual value Ch.2 <-> Data Pointer/CurrentActualValues[1]
//     Term 37 (AT2002-0250)/CC Inputs/Current actual value Ch.3 <-> Data Pointer/CurrentActualValues[2]
//     Term 37 (AT2002-0250)/CC Inputs/Current actual value Ch.4 <-> Data Pointer/CurrentActualValues[3]
//     Term 37 (AT2002-0250)/CC Inputs/Current actual value Ch.5 <-> Data Pointer/CurrentActualValues[4]
//     Term 37 (AT2002-0250)/CC Inputs/Current actual value Ch.6 <-> Data Pointer/CurrentActualValues[5]
//     Term 37 (AT2002-0250)/CC Inputs/Current actual value Ch.7 <-> Data Pointer/CurrentActualValues[6]
//     Term 37 (AT2002-0250)/CC Inputs/Current actual value Ch.8 <-> Data Pointer/CurrentActualValues[7]
//     Term 37 (AT2002-0250)/CC Inputs/Current actual value Ch.9 <-> Data Pointer/CurrentActualValues[8]
//     Term 37 (AT2002-0250)/CC Inputs/Status <-> Data Pointer/Status
//     Term 37 (AT2002-0250)/CC Outputs/Control <-> Data Pointer/Control
//     Term 37 (AT2002-0250)/CC Outputs/Current setpoint value Ch.1 <-> Data Pointer/CurrentSetpointValues[0]
//     Term 37 (AT2002-0250)/CC Outputs/Current setpoint value Ch.10 <-> Data Pointer/CurrentSetpointValues[9]
//     Term 37 (AT2002-0250)/CC Outputs/Current setpoint value Ch.11 <-> Data Pointer/CurrentSetpointValues[10]
//     Term 37 (AT2002-0250)/CC Outputs/Current setpoint value Ch.12 <-> Data Pointer/CurrentSetpointValues[11]
//     Term 37 (AT2002-0250)/CC Outputs/Current setpoint value Ch.13 <-> Data Pointer/CurrentSetpointValues[12]
//     Term 37 (AT2002-0250)/CC Outputs/Current setpoint value Ch.14 <-> Data Pointer/CurrentSetpointValues[13]
//     Term 37 (AT2002-0250)/CC Outputs/Current setpoint value Ch.15 <-> Data Pointer/CurrentSetpointValues[14]
//     Term 37 (AT2002-0250)/CC Outputs/Current setpoint value Ch.2 <-> Data Pointer/CurrentSetpointValues[1]
//     Term 37 (AT2002-0250)/CC Outputs/Current setpoint value Ch.3 <-> Data Pointer/CurrentSetpointValues[2]
//     Term 37 (AT2002-0250)/CC Outputs/Current setpoint value Ch.4 <-> Data Pointer/CurrentSetpointValues[3]
//     Term 37 (AT2002-0250)/CC Outputs/Current setpoint value Ch.5 <-> Data Pointer/CurrentSetpointValues[4]
//     Term 37 (AT2002-0250)/CC Outputs/Current setpoint value Ch.6 <-> Data Pointer/CurrentSetpointValues[5]
//     Term 37 (AT2002-0250)/CC Outputs/Current setpoint value Ch.7 <-> Data Pointer/CurrentSetpointValues[6]
//     Term 37 (AT2002-0250)/CC Outputs/Current setpoint value Ch.8 <-> Data Pointer/CurrentSetpointValues[7]
//     Term 37 (AT2002-0250)/CC Outputs/Current setpoint value Ch.9 <-> Data Pointer/CurrentSetpointValues[8]
//     Term 37 (AT2002-0250)/Term 38 (AT2002-5250)/FB Inputs/Value Channel 01 <-> Data Pointer/RawPositionValues[0]
//     Term 37 (AT2002-0250)/Term 38 (AT2002-5250)/FB Inputs/Value Channel 02 <-> Data Pointer/RawPositionValues[1]
//     Term 37 (AT2002-0250)/Term 38 (AT2002-5250)/FB Inputs/Value Channel 03 <-> Data Pointer/RawPositionValues[2]
//     Term 37 (AT2002-0250)/Term 38 (AT2002-5250)/FB Inputs/Value Channel 04 <-> Data Pointer/RawPositionValues[3]
//     Term 37 (AT2002-0250)/Term 38 (AT2002-5250)/FB Inputs/Value Channel 05 <-> Data Pointer/RawPositionValues[4]
//     Term 37 (AT2002-0250)/Term 38 (AT2002-5250)/FB Inputs/Value Channel 06 <-> Data Pointer/RawPositionValues[5]
//     Term 37 (AT2002-0250)/Term 38 (AT2002-5250)/FB Inputs/Value Channel 07 <-> Data Pointer/RawPositionValues[6]
//     Term 37 (AT2002-0250)/Term 38 (AT2002-5250)/FB Inputs/Value Channel 08 <-> Data Pointer/RawPositionValues[7]
//     Term 37 (AT2002-0250)/Term 38 (AT2002-5250)/FB Inputs/Value Channel 09 <-> Data Pointer/RawPositionValues[8]
//     Term 37 (AT2002-0250)/Term 38 (AT2002-5250)/FB Inputs/Value Channel 10 <-> Data Pointer/RawPositionValues[9]
//     Term 37 (AT2002-0250)/Term 38 (AT2002-5250)/FB Inputs/Value Channel 11 <-> Data Pointer/RawPositionValues[10]
//     Term 37 (AT2002-0250)/Term 38 (AT2002-5250)/FB Inputs/Value Channel 12 <-> Data Pointer/RawPositionValues[11]
//     Term 37 (AT2002-0250)/Term 38 (AT2002-5250)/FB Inputs/Value Channel 13 <-> Data Pointer/RawPositionValues[12]
//     Term 37 (AT2002-0250)/Term 38 (AT2002-5250)/FB Inputs/Value Channel 14 <-> Data Pointer/RawPositionValues[13]
//     Term 37 (AT2002-0250)/Term 38 (AT2002-5250)/FB Inputs/Value Channel 15 <-> Data Pointer/RawPositionValues[14]
//     Term 37 (AT2002-0250)/Term 38 (AT2002-5250)/FB Inputs/Value Channel 16 <-> Data Pointer/RawPositionValues[15]
//     Term 37 (AT2002-0250)/Term 38 (AT2002-5250)/FB Inputs/Value Channel 17 <-> Data Pointer/RawPositionValues[16]
//     Term 37 (AT2002-0250)/Term 38 (AT2002-5250)/FB Inputs/Value Channel 18 <-> Data Pointer/RawPositionValues[17]
//     Term 37 (AT2002-0250)/Term 38 (AT2002-5250)/FB Inputs/Value Channel 19 <-> Data Pointer/RawPositionValues[18]
//     Term 37 (AT2002-0250)/Term 38 (AT2002-5250)/FB Inputs/Value Channel 20 <-> Data Pointer/RawPositionValues[19]
//     Term 37 (AT2002-0250)/Term 38 (AT2002-5250)/FB Inputs/Value Channel 21 <-> Data Pointer/RawPositionValues[20]
//     Term 37 (AT2002-0250)/Term 38 (AT2002-5250)/FB Inputs/Value Channel 22 <-> Data Pointer/RawPositionValues[21]
//     Term 37 (AT2002-0250)/Term 38 (AT2002-5250)/FB Inputs/Value Channel 23 <-> Data Pointer/RawPositionValues[22]
//     Term 37 (AT2002-0250)/Term 38 (AT2002-5250)/FB Inputs/Value Channel 24 <-> Data Pointer/RawPositionValues[23]
//     Term 37 (AT2002-0250)/Term 38 (AT2002-5250)/FB Inputs/Value Channel 25 <-> Data Pointer/RawPositionValues[24]
//     Term 37 (AT2002-0250)/Term 38 (AT2002-5250)/FB Inputs/Value Channel 26 <-> Data Pointer/RawPositionValues[25]
//     Term 37 (AT2002-0250)/Term 38 (AT2002-5250)/FB Inputs/Value Channel 27 <-> Data Pointer/RawPositionValues[26]
//     Term 37 (AT2002-0250)/Term 38 (AT2002-5250)/FB Inputs/Value Channel 28 <-> Data Pointer/RawPositionValues[27]
//     Term 37 (AT2002-0250)/Term 38 (AT2002-5250)/FB Inputs/Value Channel 29 <-> Data Pointer/RawPositionValues[28]
//     Term 37 (AT2002-0250)/Term 38 (AT2002-5250)/FB Inputs/Value Channel 30 <-> Data Pointer/RawPositionValues[29]
//     Term 37 (AT2002-0250)/Term 38 (AT2002-5250)/FB Inputs/Value Channel 31 <-> Data Pointer/RawPositionValues[30]
//     Term 37 (AT2002-0250)/Term 38 (AT2002-5250)/FB Inputs/Value Channel 32 <-> Data Pointer/RawPositionValues[31]
//   Device 18 <-> TcCOM Objects/XTS ProcessingUnit 1/Part 1/Module 20
//     Term 39 (AT2000-0250)/CC Inputs/Current actual value Ch.1 <-> Data Pointer/CurrentActualValues[0]
//     Term 39 (AT2000-0250)/CC Inputs/Current actual value Ch.10 <-> Data Pointer/CurrentActualValues[9]
//     Term 39 (AT2000-0250)/CC Inputs/Current actual value Ch.11 <-> Data Pointer/CurrentActualValues[10]
//     Term 39 (AT2000-0250)/CC Inputs/Current actual value Ch.12 <-> Data Pointer/CurrentActualValues[11]
//     Term 39 (AT2000-0250)/CC Inputs/Current actual value Ch.13 <-> Data Pointer/CurrentActualValues[12]
//     Term 39 (AT2000-0250)/CC Inputs/Current actual value Ch.14 <-> Data Pointer/CurrentActualValues[13]
//     Term 39 (AT2000-0250)/CC Inputs/Current actual value Ch.15 <-> Data Pointer/CurrentActualValues[14]
//     Term 39 (AT2000-0250)/CC Inputs/Current actual value Ch.2 <-> Data Pointer/CurrentActualValues[1]
//     Term 39 (AT2000-0250)/CC Inputs/Current actual value Ch.3 <-> Data Pointer/CurrentActualValues[2]
//     Term 39 (AT2000-0250)/CC Inputs/Current actual value Ch.4 <-> Data Pointer/CurrentActualValues[3]
//     Term 39 (AT2000-0250)/CC Inputs/Current actual value Ch.5 <-> Data Pointer/CurrentActualValues[4]
//     Term 39 (AT2000-0250)/CC Inputs/Current actual value Ch.6 <-> Data Pointer/CurrentActualValues[5]
//     Term 39 (AT2000-0250)/CC Inputs/Current actual value Ch.7 <-> Data Pointer/CurrentActualValues[6]
//     Term 39 (AT2000-0250)/CC Inputs/Current actual value Ch.8 <-> Data Pointer/CurrentActualValues[7]
//     Term 39 (AT2000-0250)/CC Inputs/Current actual value Ch.9 <-> Data Pointer/CurrentActualValues[8]
//     Term 39 (AT2000-0250)/CC Inputs/Status <-> Data Pointer/Status
//     Term 39 (AT2000-0250)/CC Outputs/Control <-> Data Pointer/Control
//     Term 39 (AT2000-0250)/CC Outputs/Current setpoint value Ch.1 <-> Data Pointer/CurrentSetpointValues[0]
//     Term 39 (AT2000-0250)/CC Outputs/Current setpoint value Ch.10 <-> Data Pointer/CurrentSetpointValues[9]
//     Term 39 (AT2000-0250)/CC Outputs/Current setpoint value Ch.11 <-> Data Pointer/CurrentSetpointValues[10]
//     Term 39 (AT2000-0250)/CC Outputs/Current setpoint value Ch.12 <-> Data Pointer/CurrentSetpointValues[11]
//     Term 39 (AT2000-0250)/CC Outputs/Current setpoint value Ch.13 <-> Data Pointer/CurrentSetpointValues[12]
//     Term 39 (AT2000-0250)/CC Outputs/Current setpoint value Ch.14 <-> Data Pointer/CurrentSetpointValues[13]
//     Term 39 (AT2000-0250)/CC Outputs/Current setpoint value Ch.15 <-> Data Pointer/CurrentSetpointValues[14]
//     Term 39 (AT2000-0250)/CC Outputs/Current setpoint value Ch.2 <-> Data Pointer/CurrentSetpointValues[1]
//     Term 39 (AT2000-0250)/CC Outputs/Current setpoint value Ch.3 <-> Data Pointer/CurrentSetpointValues[2]
//     Term 39 (AT2000-0250)/CC Outputs/Current setpoint value Ch.4 <-> Data Pointer/CurrentSetpointValues[3]
//     Term 39 (AT2000-0250)/CC Outputs/Current setpoint value Ch.5 <-> Data Pointer/CurrentSetpointValues[4]
//     Term 39 (AT2000-0250)/CC Outputs/Current setpoint value Ch.6 <-> Data Pointer/CurrentSetpointValues[5]
//     Term 39 (AT2000-0250)/CC Outputs/Current setpoint value Ch.7 <-> Data Pointer/CurrentSetpointValues[6]
//     Term 39 (AT2000-0250)/CC Outputs/Current setpoint value Ch.8 <-> Data Pointer/CurrentSetpointValues[7]
//     Term 39 (AT2000-0250)/CC Outputs/Current setpoint value Ch.9 <-> Data Pointer/CurrentSetpointValues[8]
//     Term 39 (AT2000-0250)/Term 40 (AT2000-5250)/FB Inputs/Value Channel 01 <-> Data Pointer/RawPositionValues[0]
//     Term 39 (AT2000-0250)/Term 40 (AT2000-5250)/FB Inputs/Value Channel 02 <-> Data Pointer/RawPositionValues[1]
//     Term 39 (AT2000-0250)/Term 40 (AT2000-5250)/FB Inputs/Value Channel 03 <-> Data Pointer/RawPositionValues[2]
//     Term 39 (AT2000-0250)/Term 40 (AT2000-5250)/FB Inputs/Value Channel 04 <-> Data Pointer/RawPositionValues[3]
//     Term 39 (AT2000-0250)/Term 40 (AT2000-5250)/FB Inputs/Value Channel 05 <-> Data Pointer/RawPositionValues[4]
//     Term 39 (AT2000-0250)/Term 40 (AT2000-5250)/FB Inputs/Value Channel 06 <-> Data Pointer/RawPositionValues[5]
//     Term 39 (AT2000-0250)/Term 40 (AT2000-5250)/FB Inputs/Value Channel 07 <-> Data Pointer/RawPositionValues[6]
//     Term 39 (AT2000-0250)/Term 40 (AT2000-5250)/FB Inputs/Value Channel 08 <-> Data Pointer/RawPositionValues[7]
//     Term 39 (AT2000-0250)/Term 40 (AT2000-5250)/FB Inputs/Value Channel 09 <-> Data Pointer/RawPositionValues[8]
//     Term 39 (AT2000-0250)/Term 40 (AT2000-5250)/FB Inputs/Value Channel 10 <-> Data Pointer/RawPositionValues[9]
//     Term 39 (AT2000-0250)/Term 40 (AT2000-5250)/FB Inputs/Value Channel 11 <-> Data Pointer/RawPositionValues[10]
//     Term 39 (AT2000-0250)/Term 40 (AT2000-5250)/FB Inputs/Value Channel 12 <-> Data Pointer/RawPositionValues[11]
//     Term 39 (AT2000-0250)/Term 40 (AT2000-5250)/FB Inputs/Value Channel 13 <-> Data Pointer/RawPositionValues[12]
//     Term 39 (AT2000-0250)/Term 40 (AT2000-5250)/FB Inputs/Value Channel 14 <-> Data Pointer/RawPositionValues[13]
//     Term 39 (AT2000-0250)/Term 40 (AT2000-5250)/FB Inputs/Value Channel 15 <-> Data Pointer/RawPositionValues[14]
//     Term 39 (AT2000-0250)/Term 40 (AT2000-5250)/FB Inputs/Value Channel 16 <-> Data Pointer/RawPositionValues[15]
//     Term 39 (AT2000-0250)/Term 40 (AT2000-5250)/FB Inputs/Value Channel 17 <-> Data Pointer/RawPositionValues[16]
//     Term 39 (AT2000-0250)/Term 40 (AT2000-5250)/FB Inputs/Value Channel 18 <-> Data Pointer/RawPositionValues[17]
//     Term 39 (AT2000-0250)/Term 40 (AT2000-5250)/FB Inputs/Value Channel 19 <-> Data Pointer/RawPositionValues[18]
//     Term 39 (AT2000-0250)/Term 40 (AT2000-5250)/FB Inputs/Value Channel 20 <-> Data Pointer/RawPositionValues[19]
//     Term 39 (AT2000-0250)/Term 40 (AT2000-5250)/FB Inputs/Value Channel 21 <-> Data Pointer/RawPositionValues[20]
//     Term 39 (AT2000-0250)/Term 40 (AT2000-5250)/FB Inputs/Value Channel 22 <-> Data Pointer/RawPositionValues[21]
//     Term 39 (AT2000-0250)/Term 40 (AT2000-5250)/FB Inputs/Value Channel 23 <-> Data Pointer/RawPositionValues[22]
//     Term 39 (AT2000-0250)/Term 40 (AT2000-5250)/FB Inputs/Value Channel 24 <-> Data Pointer/RawPositionValues[23]
//     Term 39 (AT2000-0250)/Term 40 (AT2000-5250)/FB Inputs/Value Channel 25 <-> Data Pointer/RawPositionValues[24]
//     Term 39 (AT2000-0250)/Term 40 (AT2000-5250)/FB Inputs/Value Channel 26 <-> Data Pointer/RawPositionValues[25]
//     Term 39 (AT2000-0250)/Term 40 (AT2000-5250)/FB Inputs/Value Channel 27 <-> Data Pointer/RawPositionValues[26]
//     Term 39 (AT2000-0250)/Term 40 (AT2000-5250)/FB Inputs/Value Channel 28 <-> Data Pointer/RawPositionValues[27]
//     Term 39 (AT2000-0250)/Term 40 (AT2000-5250)/FB Inputs/Value Channel 29 <-> Data Pointer/RawPositionValues[28]
//     Term 39 (AT2000-0250)/Term 40 (AT2000-5250)/FB Inputs/Value Channel 30 <-> Data Pointer/RawPositionValues[29]
//     Term 39 (AT2000-0250)/Term 40 (AT2000-5250)/FB Inputs/Value Channel 31 <-> Data Pointer/RawPositionValues[30]
//     Term 39 (AT2000-0250)/Term 40 (AT2000-5250)/FB Inputs/Value Channel 32 <-> Data Pointer/RawPositionValues[31]
//   Device 18 <-> TcCOM Objects/XTS ProcessingUnit 1/Part 1/Module 21
//     Term 41 (AT2000-0250)/CC Inputs/Current actual value Ch.1 <-> Data Pointer/CurrentActualValues[0]
//     Term 41 (AT2000-0250)/CC Inputs/Current actual value Ch.10 <-> Data Pointer/CurrentActualValues[9]
//     Term 41 (AT2000-0250)/CC Inputs/Current actual value Ch.11 <-> Data Pointer/CurrentActualValues[10]
//     Term 41 (AT2000-0250)/CC Inputs/Current actual value Ch.12 <-> Data Pointer/CurrentActualValues[11]
//     Term 41 (AT2000-0250)/CC Inputs/Current actual value Ch.13 <-> Data Pointer/CurrentActualValues[12]
//     Term 41 (AT2000-0250)/CC Inputs/Current actual value Ch.14 <-> Data Pointer/CurrentActualValues[13]
//     Term 41 (AT2000-0250)/CC Inputs/Current actual value Ch.15 <-> Data Pointer/CurrentActualValues[14]
//     Term 41 (AT2000-0250)/CC Inputs/Current actual value Ch.2 <-> Data Pointer/CurrentActualValues[1]
//     Term 41 (AT2000-0250)/CC Inputs/Current actual value Ch.3 <-> Data Pointer/CurrentActualValues[2]
//     Term 41 (AT2000-0250)/CC Inputs/Current actual value Ch.4 <-> Data Pointer/CurrentActualValues[3]
//     Term 41 (AT2000-0250)/CC Inputs/Current actual value Ch.5 <-> Data Pointer/CurrentActualValues[4]
//     Term 41 (AT2000-0250)/CC Inputs/Current actual value Ch.6 <-> Data Pointer/CurrentActualValues[5]
//     Term 41 (AT2000-0250)/CC Inputs/Current actual value Ch.7 <-> Data Pointer/CurrentActualValues[6]
//     Term 41 (AT2000-0250)/CC Inputs/Current actual value Ch.8 <-> Data Pointer/CurrentActualValues[7]
//     Term 41 (AT2000-0250)/CC Inputs/Current actual value Ch.9 <-> Data Pointer/CurrentActualValues[8]
//     Term 41 (AT2000-0250)/CC Inputs/Status <-> Data Pointer/Status
//     Term 41 (AT2000-0250)/CC Outputs/Control <-> Data Pointer/Control
//     Term 41 (AT2000-0250)/CC Outputs/Current setpoint value Ch.1 <-> Data Pointer/CurrentSetpointValues[0]
//     Term 41 (AT2000-0250)/CC Outputs/Current setpoint value Ch.10 <-> Data Pointer/CurrentSetpointValues[9]
//     Term 41 (AT2000-0250)/CC Outputs/Current setpoint value Ch.11 <-> Data Pointer/CurrentSetpointValues[10]
//     Term 41 (AT2000-0250)/CC Outputs/Current setpoint value Ch.12 <-> Data Pointer/CurrentSetpointValues[11]
//     Term 41 (AT2000-0250)/CC Outputs/Current setpoint value Ch.13 <-> Data Pointer/CurrentSetpointValues[12]
//     Term 41 (AT2000-0250)/CC Outputs/Current setpoint value Ch.14 <-> Data Pointer/CurrentSetpointValues[13]
//     Term 41 (AT2000-0250)/CC Outputs/Current setpoint value Ch.15 <-> Data Pointer/CurrentSetpointValues[14]
//     Term 41 (AT2000-0250)/CC Outputs/Current setpoint value Ch.2 <-> Data Pointer/CurrentSetpointValues[1]
//     Term 41 (AT2000-0250)/CC Outputs/Current setpoint value Ch.3 <-> Data Pointer/CurrentSetpointValues[2]
//     Term 41 (AT2000-0250)/CC Outputs/Current setpoint value Ch.4 <-> Data Pointer/CurrentSetpointValues[3]
//     Term 41 (AT2000-0250)/CC Outputs/Current setpoint value Ch.5 <-> Data Pointer/CurrentSetpointValues[4]
//     Term 41 (AT2000-0250)/CC Outputs/Current setpoint value Ch.6 <-> Data Pointer/CurrentSetpointValues[5]
//     Term 41 (AT2000-0250)/CC Outputs/Current setpoint value Ch.7 <-> Data Pointer/CurrentSetpointValues[6]
//     Term 41 (AT2000-0250)/CC Outputs/Current setpoint value Ch.8 <-> Data Pointer/CurrentSetpointValues[7]
//     Term 41 (AT2000-0250)/CC Outputs/Current setpoint value Ch.9 <-> Data Pointer/CurrentSetpointValues[8]
//     Term 41 (AT2000-0250)/Term 42 (AT2000-5250)/FB Inputs/Value Channel 01 <-> Data Pointer/RawPositionValues[0]
//     Term 41 (AT2000-0250)/Term 42 (AT2000-5250)/FB Inputs/Value Channel 02 <-> Data Pointer/RawPositionValues[1]
//     Term 41 (AT2000-0250)/Term 42 (AT2000-5250)/FB Inputs/Value Channel 03 <-> Data Pointer/RawPositionValues[2]
//     Term 41 (AT2000-0250)/Term 42 (AT2000-5250)/FB Inputs/Value Channel 04 <-> Data Pointer/RawPositionValues[3]
//     Term 41 (AT2000-0250)/Term 42 (AT2000-5250)/FB Inputs/Value Channel 05 <-> Data Pointer/RawPositionValues[4]
//     Term 41 (AT2000-0250)/Term 42 (AT2000-5250)/FB Inputs/Value Channel 06 <-> Data Pointer/RawPositionValues[5]
//     Term 41 (AT2000-0250)/Term 42 (AT2000-5250)/FB Inputs/Value Channel 07 <-> Data Pointer/RawPositionValues[6]
//     Term 41 (AT2000-0250)/Term 42 (AT2000-5250)/FB Inputs/Value Channel 08 <-> Data Pointer/RawPositionValues[7]
//     Term 41 (AT2000-0250)/Term 42 (AT2000-5250)/FB Inputs/Value Channel 09 <-> Data Pointer/RawPositionValues[8]
//     Term 41 (AT2000-0250)/Term 42 (AT2000-5250)/FB Inputs/Value Channel 10 <-> Data Pointer/RawPositionValues[9]
//     Term 41 (AT2000-0250)/Term 42 (AT2000-5250)/FB Inputs/Value Channel 11 <-> Data Pointer/RawPositionValues[10]
//     Term 41 (AT2000-0250)/Term 42 (AT2000-5250)/FB Inputs/Value Channel 12 <-> Data Pointer/RawPositionValues[11]
//     Term 41 (AT2000-0250)/Term 42 (AT2000-5250)/FB Inputs/Value Channel 13 <-> Data Pointer/RawPositionValues[12]
//     Term 41 (AT2000-0250)/Term 42 (AT2000-5250)/FB Inputs/Value Channel 14 <-> Data Pointer/RawPositionValues[13]
//     Term 41 (AT2000-0250)/Term 42 (AT2000-5250)/FB Inputs/Value Channel 15 <-> Data Pointer/RawPositionValues[14]
//     Term 41 (AT2000-0250)/Term 42 (AT2000-5250)/FB Inputs/Value Channel 16 <-> Data Pointer/RawPositionValues[15]
//     Term 41 (AT2000-0250)/Term 42 (AT2000-5250)/FB Inputs/Value Channel 17 <-> Data Pointer/RawPositionValues[16]
//     Term 41 (AT2000-0250)/Term 42 (AT2000-5250)/FB Inputs/Value Channel 18 <-> Data Pointer/RawPositionValues[17]
//     Term 41 (AT2000-0250)/Term 42 (AT2000-5250)/FB Inputs/Value Channel 19 <-> Data Pointer/RawPositionValues[18]
//     Term 41 (AT2000-0250)/Term 42 (AT2000-5250)/FB Inputs/Value Channel 20 <-> Data Pointer/RawPositionValues[19]
//     Term 41 (AT2000-0250)/Term 42 (AT2000-5250)/FB Inputs/Value Channel 21 <-> Data Pointer/RawPositionValues[20]
//     Term 41 (AT2000-0250)/Term 42 (AT2000-5250)/FB Inputs/Value Channel 22 <-> Data Pointer/RawPositionValues[21]
//     Term 41 (AT2000-0250)/Term 42 (AT2000-5250)/FB Inputs/Value Channel 23 <-> Data Pointer/RawPositionValues[22]
//     Term 41 (AT2000-0250)/Term 42 (AT2000-5250)/FB Inputs/Value Channel 24 <-> Data Pointer/RawPositionValues[23]
//     Term 41 (AT2000-0250)/Term 42 (AT2000-5250)/FB Inputs/Value Channel 25 <-> Data Pointer/RawPositionValues[24]
//     Term 41 (AT2000-0250)/Term 42 (AT2000-5250)/FB Inputs/Value Channel 26 <-> Data Pointer/RawPositionValues[25]
//     Term 41 (AT2000-0250)/Term 42 (AT2000-5250)/FB Inputs/Value Channel 27 <-> Data Pointer/RawPositionValues[26]
//     Term 41 (AT2000-0250)/Term 42 (AT2000-5250)/FB Inputs/Value Channel 28 <-> Data Pointer/RawPositionValues[27]
//     Term 41 (AT2000-0250)/Term 42 (AT2000-5250)/FB Inputs/Value Channel 29 <-> Data Pointer/RawPositionValues[28]
//     Term 41 (AT2000-0250)/Term 42 (AT2000-5250)/FB Inputs/Value Channel 30 <-> Data Pointer/RawPositionValues[29]
//     Term 41 (AT2000-0250)/Term 42 (AT2000-5250)/FB Inputs/Value Channel 31 <-> Data Pointer/RawPositionValues[30]
//     Term 41 (AT2000-0250)/Term 42 (AT2000-5250)/FB Inputs/Value Channel 32 <-> Data Pointer/RawPositionValues[31]
//   Device 18 <-> TcCOM Objects/XTS ProcessingUnit 1/Part 1/Module 22
//     Term 43 (AT2000-0250)/CC Inputs/Current actual value Ch.1 <-> Data Pointer/CurrentActualValues[0]
//     Term 43 (AT2000-0250)/CC Inputs/Current actual value Ch.10 <-> Data Pointer/CurrentActualValues[9]
//     Term 43 (AT2000-0250)/CC Inputs/Current actual value Ch.11 <-> Data Pointer/CurrentActualValues[10]
//     Term 43 (AT2000-0250)/CC Inputs/Current actual value Ch.12 <-> Data Pointer/CurrentActualValues[11]
//     Term 43 (AT2000-0250)/CC Inputs/Current actual value Ch.13 <-> Data Pointer/CurrentActualValues[12]
//     Term 43 (AT2000-0250)/CC Inputs/Current actual value Ch.14 <-> Data Pointer/CurrentActualValues[13]
//     Term 43 (AT2000-0250)/CC Inputs/Current actual value Ch.15 <-> Data Pointer/CurrentActualValues[14]
//     Term 43 (AT2000-0250)/CC Inputs/Current actual value Ch.2 <-> Data Pointer/CurrentActualValues[1]
//     Term 43 (AT2000-0250)/CC Inputs/Current actual value Ch.3 <-> Data Pointer/CurrentActualValues[2]
//     Term 43 (AT2000-0250)/CC Inputs/Current actual value Ch.4 <-> Data Pointer/CurrentActualValues[3]
//     Term 43 (AT2000-0250)/CC Inputs/Current actual value Ch.5 <-> Data Pointer/CurrentActualValues[4]
//     Term 43 (AT2000-0250)/CC Inputs/Current actual value Ch.6 <-> Data Pointer/CurrentActualValues[5]
//     Term 43 (AT2000-0250)/CC Inputs/Current actual value Ch.7 <-> Data Pointer/CurrentActualValues[6]
//     Term 43 (AT2000-0250)/CC Inputs/Current actual value Ch.8 <-> Data Pointer/CurrentActualValues[7]
//     Term 43 (AT2000-0250)/CC Inputs/Current actual value Ch.9 <-> Data Pointer/CurrentActualValues[8]
//     Term 43 (AT2000-0250)/CC Inputs/Status <-> Data Pointer/Status
//     Term 43 (AT2000-0250)/CC Outputs/Control <-> Data Pointer/Control
//     Term 43 (AT2000-0250)/CC Outputs/Current setpoint value Ch.1 <-> Data Pointer/CurrentSetpointValues[0]
//     Term 43 (AT2000-0250)/CC Outputs/Current setpoint value Ch.10 <-> Data Pointer/CurrentSetpointValues[9]
//     Term 43 (AT2000-0250)/CC Outputs/Current setpoint value Ch.11 <-> Data Pointer/CurrentSetpointValues[10]
//     Term 43 (AT2000-0250)/CC Outputs/Current setpoint value Ch.12 <-> Data Pointer/CurrentSetpointValues[11]
//     Term 43 (AT2000-0250)/CC Outputs/Current setpoint value Ch.13 <-> Data Pointer/CurrentSetpointValues[12]
//     Term 43 (AT2000-0250)/CC Outputs/Current setpoint value Ch.14 <-> Data Pointer/CurrentSetpointValues[13]
//     Term 43 (AT2000-0250)/CC Outputs/Current setpoint value Ch.15 <-> Data Pointer/CurrentSetpointValues[14]
//     Term 43 (AT2000-0250)/CC Outputs/Current setpoint value Ch.2 <-> Data Pointer/CurrentSetpointValues[1]
//     Term 43 (AT2000-0250)/CC Outputs/Current setpoint value Ch.3 <-> Data Pointer/CurrentSetpointValues[2]
//     Term 43 (AT2000-0250)/CC Outputs/Current setpoint value Ch.4 <-> Data Pointer/CurrentSetpointValues[3]
//     Term 43 (AT2000-0250)/CC Outputs/Current setpoint value Ch.5 <-> Data Pointer/CurrentSetpointValues[4]
//     Term 43 (AT2000-0250)/CC Outputs/Current setpoint value Ch.6 <-> Data Pointer/CurrentSetpointValues[5]
//     Term 43 (AT2000-0250)/CC Outputs/Current setpoint value Ch.7 <-> Data Pointer/CurrentSetpointValues[6]
//     Term 43 (AT2000-0250)/CC Outputs/Current setpoint value Ch.8 <-> Data Pointer/CurrentSetpointValues[7]
//     Term 43 (AT2000-0250)/CC Outputs/Current setpoint value Ch.9 <-> Data Pointer/CurrentSetpointValues[8]
//     Term 43 (AT2000-0250)/Term 44 (AT2000-5250)/FB Inputs/Value Channel 01 <-> Data Pointer/RawPositionValues[0]
//     Term 43 (AT2000-0250)/Term 44 (AT2000-5250)/FB Inputs/Value Channel 02 <-> Data Pointer/RawPositionValues[1]
//     Term 43 (AT2000-0250)/Term 44 (AT2000-5250)/FB Inputs/Value Channel 03 <-> Data Pointer/RawPositionValues[2]
//     Term 43 (AT2000-0250)/Term 44 (AT2000-5250)/FB Inputs/Value Channel 04 <-> Data Pointer/RawPositionValues[3]
//     Term 43 (AT2000-0250)/Term 44 (AT2000-5250)/FB Inputs/Value Channel 05 <-> Data Pointer/RawPositionValues[4]
//     Term 43 (AT2000-0250)/Term 44 (AT2000-5250)/FB Inputs/Value Channel 06 <-> Data Pointer/RawPositionValues[5]
//     Term 43 (AT2000-0250)/Term 44 (AT2000-5250)/FB Inputs/Value Channel 07 <-> Data Pointer/RawPositionValues[6]
//     Term 43 (AT2000-0250)/Term 44 (AT2000-5250)/FB Inputs/Value Channel 08 <-> Data Pointer/RawPositionValues[7]
//     Term 43 (AT2000-0250)/Term 44 (AT2000-5250)/FB Inputs/Value Channel 09 <-> Data Pointer/RawPositionValues[8]
//     Term 43 (AT2000-0250)/Term 44 (AT2000-5250)/FB Inputs/Value Channel 10 <-> Data Pointer/RawPositionValues[9]
//     Term 43 (AT2000-0250)/Term 44 (AT2000-5250)/FB Inputs/Value Channel 11 <-> Data Pointer/RawPositionValues[10]
//     Term 43 (AT2000-0250)/Term 44 (AT2000-5250)/FB Inputs/Value Channel 12 <-> Data Pointer/RawPositionValues[11]
//     Term 43 (AT2000-0250)/Term 44 (AT2000-5250)/FB Inputs/Value Channel 13 <-> Data Pointer/RawPositionValues[12]
//     Term 43 (AT2000-0250)/Term 44 (AT2000-5250)/FB Inputs/Value Channel 14 <-> Data Pointer/RawPositionValues[13]
//     Term 43 (AT2000-0250)/Term 44 (AT2000-5250)/FB Inputs/Value Channel 15 <-> Data Pointer/RawPositionValues[14]
//     Term 43 (AT2000-0250)/Term 44 (AT2000-5250)/FB Inputs/Value Channel 16 <-> Data Pointer/RawPositionValues[15]
//     Term 43 (AT2000-0250)/Term 44 (AT2000-5250)/FB Inputs/Value Channel 17 <-> Data Pointer/RawPositionValues[16]
//     Term 43 (AT2000-0250)/Term 44 (AT2000-5250)/FB Inputs/Value Channel 18 <-> Data Pointer/RawPositionValues[17]
//     Term 43 (AT2000-0250)/Term 44 (AT2000-5250)/FB Inputs/Value Channel 19 <-> Data Pointer/RawPositionValues[18]
//     Term 43 (AT2000-0250)/Term 44 (AT2000-5250)/FB Inputs/Value Channel 20 <-> Data Pointer/RawPositionValues[19]
//     Term 43 (AT2000-0250)/Term 44 (AT2000-5250)/FB Inputs/Value Channel 21 <-> Data Pointer/RawPositionValues[20]
//     Term 43 (AT2000-0250)/Term 44 (AT2000-5250)/FB Inputs/Value Channel 22 <-> Data Pointer/RawPositionValues[21]
//     Term 43 (AT2000-0250)/Term 44 (AT2000-5250)/FB Inputs/Value Channel 23 <-> Data Pointer/RawPositionValues[22]
//     Term 43 (AT2000-0250)/Term 44 (AT2000-5250)/FB Inputs/Value Channel 24 <-> Data Pointer/RawPositionValues[23]
//     Term 43 (AT2000-0250)/Term 44 (AT2000-5250)/FB Inputs/Value Channel 25 <-> Data Pointer/RawPositionValues[24]
//     Term 43 (AT2000-0250)/Term 44 (AT2000-5250)/FB Inputs/Value Channel 26 <-> Data Pointer/RawPositionValues[25]
//     Term 43 (AT2000-0250)/Term 44 (AT2000-5250)/FB Inputs/Value Channel 27 <-> Data Pointer/RawPositionValues[26]
//     Term 43 (AT2000-0250)/Term 44 (AT2000-5250)/FB Inputs/Value Channel 28 <-> Data Pointer/RawPositionValues[27]
//     Term 43 (AT2000-0250)/Term 44 (AT2000-5250)/FB Inputs/Value Channel 29 <-> Data Pointer/RawPositionValues[28]
//     Term 43 (AT2000-0250)/Term 44 (AT2000-5250)/FB Inputs/Value Channel 30 <-> Data Pointer/RawPositionValues[29]
//     Term 43 (AT2000-0250)/Term 44 (AT2000-5250)/FB Inputs/Value Channel 31 <-> Data Pointer/RawPositionValues[30]
//     Term 43 (AT2000-0250)/Term 44 (AT2000-5250)/FB Inputs/Value Channel 32 <-> Data Pointer/RawPositionValues[31]
//   Device 18 <-> TcCOM Objects/XTS ProcessingUnit 1/Part 1/Module 23
//     Term 45 (AT2000-0250)/CC Inputs/Current actual value Ch.1 <-> Data Pointer/CurrentActualValues[0]
//     Term 45 (AT2000-0250)/CC Inputs/Current actual value Ch.10 <-> Data Pointer/CurrentActualValues[9]
//     Term 45 (AT2000-0250)/CC Inputs/Current actual value Ch.11 <-> Data Pointer/CurrentActualValues[10]
//     Term 45 (AT2000-0250)/CC Inputs/Current actual value Ch.12 <-> Data Pointer/CurrentActualValues[11]
//     Term 45 (AT2000-0250)/CC Inputs/Current actual value Ch.13 <-> Data Pointer/CurrentActualValues[12]
//     Term 45 (AT2000-0250)/CC Inputs/Current actual value Ch.14 <-> Data Pointer/CurrentActualValues[13]
//     Term 45 (AT2000-0250)/CC Inputs/Current actual value Ch.15 <-> Data Pointer/CurrentActualValues[14]
//     Term 45 (AT2000-0250)/CC Inputs/Current actual value Ch.2 <-> Data Pointer/CurrentActualValues[1]
//     Term 45 (AT2000-0250)/CC Inputs/Current actual value Ch.3 <-> Data Pointer/CurrentActualValues[2]
//     Term 45 (AT2000-0250)/CC Inputs/Current actual value Ch.4 <-> Data Pointer/CurrentActualValues[3]
//     Term 45 (AT2000-0250)/CC Inputs/Current actual value Ch.5 <-> Data Pointer/CurrentActualValues[4]
//     Term 45 (AT2000-0250)/CC Inputs/Current actual value Ch.6 <-> Data Pointer/CurrentActualValues[5]
//     Term 45 (AT2000-0250)/CC Inputs/Current actual value Ch.7 <-> Data Pointer/CurrentActualValues[6]
//     Term 45 (AT2000-0250)/CC Inputs/Current actual value Ch.8 <-> Data Pointer/CurrentActualValues[7]
//     Term 45 (AT2000-0250)/CC Inputs/Current actual value Ch.9 <-> Data Pointer/CurrentActualValues[8]
//     Term 45 (AT2000-0250)/CC Inputs/Status <-> Data Pointer/Status
